Yaskawa INFORM job: A_ROOF_UPPER_0614_2_PAINT_60.JBI

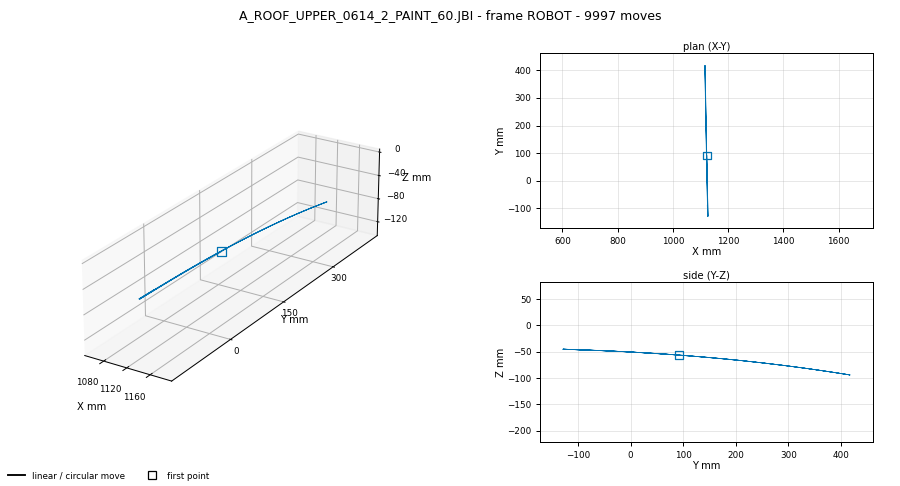
[picture p0: tool path of A_ROOF_UPPER_0614_2_PAINT_60.JBI in frame ROBOT, 9997 of 9997 moves have a stored position in this frame; points joined in program order, loops and branches not executed]
/JOB
//NAME A_ROOF_UPPER_0614_2_PAINT60
//POS
///NPOS 9997,0,0,0,0,0
///TOOL 1
///USER 0
///POSTYPE ROBOT
///RECTAN
///RCONF 1,0,0,0,0,0,0,0,0,0,0,0,0,0,0,0,0,0,0,0,0,0,0,0
C00000=1122.941,91.660,-56.179,-179.955,7.882,149.484
C00001=1122.946,91.411,-56.161,-179.956,7.878,149.483
C00002=1122.951,91.162,-56.142,-179.958,7.874,149.483
C00003=1122.955,90.913,-56.124,-179.959,7.870,149.482
C00004=1122.960,90.663,-56.106,-179.961,7.866,149.482
C00005=1122.965,90.414,-56.088,-179.962,7.862,149.481
C00006=1122.969,90.199,-56.073,-179.963,7.859,149.481
C00007=1122.974,89.984,-56.057,-179.965,7.855,149.480
C00008=1122.978,89.770,-56.041,-179.966,7.852,149.480
C00009=1122.982,89.556,-56.025,-179.967,7.849,149.480
C00010=1122.986,89.341,-56.010,-179.969,7.845,149.479
C00011=1122.990,89.126,-55.995,-179.970,7.842,149.479
C00012=1122.994,88.912,-55.978,-179.971,7.839,149.478
C00013=1122.998,88.697,-55.963,-179.972,7.835,149.478
C00014=1123.004,88.448,-55.944,-179.974,7.831,149.478
C00015=1123.009,88.199,-55.926,-179.975,7.828,149.477
C00016=1123.013,87.950,-55.908,-179.976,7.824,149.477
C00017=1123.018,87.700,-55.891,-179.978,7.820,149.476
C00018=1123.023,87.450,-55.872,-179.979,7.816,149.476
C00019=1123.028,87.201,-55.854,-179.980,7.812,149.475
C00020=1123.033,86.952,-55.836,-179.981,7.809,149.475
C00021=1123.037,86.703,-55.818,-179.983,7.805,149.474
C00022=1123.042,86.454,-55.800,-179.984,7.800,149.474
C00023=1123.048,86.204,-55.783,-179.986,7.797,149.473
C00024=1123.052,85.955,-55.765,-179.987,7.793,149.473
C00025=1123.057,85.706,-55.747,-179.988,7.789,149.472
C00026=1123.062,85.456,-55.729,-179.989,7.785,149.472
C00027=1123.067,85.207,-55.711,-179.991,7.781,149.471
C00028=1123.072,84.957,-55.693,-179.992,7.778,149.471
C00029=1123.076,84.708,-55.675,-179.993,7.774,149.470
C00030=1123.081,84.459,-55.657,-179.995,7.770,149.470
C00031=1123.086,84.210,-55.639,-179.996,7.766,149.469
C00032=1123.091,83.960,-55.622,-179.997,7.763,149.469
C00033=1123.096,83.711,-55.604,-179.998,7.759,149.468
C00034=1123.101,83.462,-55.586,-180.000,7.755,149.468
C00035=1123.105,83.213,-55.568,180.000,7.751,149.467
C00036=1123.110,82.964,-55.550,179.998,7.747,149.466
C00037=1123.116,82.714,-55.533,179.997,7.743,149.466
C00038=1123.120,82.465,-55.515,179.996,7.740,149.465
C00039=1123.125,82.216,-55.497,179.995,7.736,149.465
C00040=1123.130,81.966,-55.479,179.994,7.732,149.464
C00041=1123.136,81.717,-55.462,179.993,7.728,149.464
C00042=1123.140,81.467,-55.443,179.991,7.725,149.463
C00043=1123.145,81.217,-55.425,179.991,7.721,149.463
C00044=1123.150,80.968,-55.407,179.989,7.717,149.462
C00045=1123.154,80.719,-55.391,179.988,7.714,149.462
C00046=1123.159,80.470,-55.373,179.987,7.710,149.461
C00047=1123.164,80.220,-55.355,179.986,7.705,149.461
C00048=1123.169,79.971,-55.338,179.985,7.702,149.460
C00049=1123.174,79.722,-55.320,179.984,7.698,149.460
C00050=1123.179,79.472,-55.302,179.983,7.695,149.459
C00051=1123.183,79.223,-55.285,179.982,7.691,149.459
C00052=1123.188,78.974,-55.267,179.981,7.687,149.458
C00053=1123.193,78.724,-55.249,179.979,7.683,149.457
C00054=1123.199,78.475,-55.232,179.979,7.680,149.457
C00055=1123.204,78.226,-55.214,179.977,7.676,149.456
C00056=1123.209,77.977,-55.197,179.977,7.672,149.456
C00057=1123.213,77.728,-55.179,179.975,7.668,149.455
C00058=1123.218,77.478,-55.161,179.975,7.665,149.455
C00059=1123.224,77.229,-55.144,179.974,7.661,149.454
C00060=1123.228,76.979,-55.126,179.973,7.658,149.454
C00061=1123.233,76.730,-55.110,179.972,7.654,149.453
C00062=1123.237,76.515,-55.094,179.971,7.650,149.453
C00063=1123.241,76.300,-55.079,179.970,7.647,149.452
C00064=1123.245,76.086,-55.063,179.968,7.643,149.452
C00065=1123.250,75.871,-55.049,179.967,7.640,149.451
C00066=1123.255,75.656,-55.034,179.966,7.637,149.451
C00067=1123.258,75.442,-55.019,179.964,7.633,149.451
C00068=1123.262,75.227,-55.004,179.963,7.630,149.450
C00069=1123.266,75.012,-54.989,179.962,7.626,149.450
C00070=1123.272,74.763,-54.971,179.960,7.622,149.449
C00071=1123.276,74.514,-54.955,179.959,7.618,149.449
C00072=1123.282,74.264,-54.937,179.958,7.615,149.448
C00073=1123.287,74.015,-54.919,179.956,7.611,149.448
C00074=1123.291,73.765,-54.903,179.955,7.607,149.447
C00075=1123.296,73.516,-54.885,179.954,7.603,149.447
C00076=1123.301,73.267,-54.867,179.952,7.599,149.446
C00077=1123.305,73.018,-54.850,179.950,7.595,149.446
C00078=1123.311,72.768,-54.833,179.949,7.591,149.445
C00079=1123.316,72.519,-54.816,179.948,7.587,149.445
C00080=1123.321,72.270,-54.798,179.946,7.583,149.444
C00081=1123.326,72.020,-54.781,179.945,7.579,149.444
C00082=1123.330,71.771,-54.765,179.944,7.575,149.443
C00083=1123.335,71.521,-54.747,179.942,7.571,149.443
C00084=1123.340,71.272,-54.729,179.940,7.567,149.442
C00085=1123.345,71.022,-54.713,179.939,7.563,149.442
C00086=1123.350,70.774,-54.695,179.938,7.559,149.441
C00087=1123.355,70.524,-54.678,179.936,7.555,149.441
C00088=1123.360,70.274,-54.661,179.935,7.551,149.441
C00089=1123.365,70.025,-54.644,179.933,7.547,149.440
C00090=1123.369,69.776,-54.626,179.932,7.543,149.439
C00091=1123.375,69.527,-54.610,179.930,7.539,149.439
C00092=1123.380,69.277,-54.593,179.929,7.535,149.439
C00093=1123.385,69.027,-54.576,179.928,7.532,149.438
C00094=1123.389,68.779,-54.558,179.927,7.528,149.438
C00095=1123.394,68.529,-54.541,179.925,7.524,149.437
C00096=1123.399,68.280,-54.525,179.924,7.519,149.436
C00097=1123.405,68.030,-54.507,179.922,7.516,149.436
C00098=1123.409,67.781,-54.491,179.921,7.512,149.436
C00099=1123.414,67.531,-54.473,179.919,7.508,149.435
C00100=1123.419,67.283,-54.456,179.918,7.503,149.435
C00101=1123.424,67.033,-54.439,179.917,7.500,149.434
C00102=1123.429,66.783,-54.422,179.915,7.496,149.434
C00103=1123.433,66.534,-54.406,179.914,7.491,149.433
C00104=1123.439,66.285,-54.389,179.912,7.487,149.433
C00105=1123.444,66.035,-54.372,179.911,7.484,149.432
C00106=1123.449,65.786,-54.355,179.910,7.479,149.432
C00107=1123.453,65.536,-54.338,179.908,7.475,149.431
C00108=1123.459,65.287,-54.321,179.907,7.471,149.431
C00109=1123.464,65.038,-54.305,179.905,7.467,149.430
C00110=1123.468,64.788,-54.288,179.904,7.463,149.430
C00111=1123.473,64.538,-54.271,179.903,7.460,149.429
C00112=1123.478,64.289,-54.255,179.902,7.456,149.429
C00113=1123.483,64.040,-54.238,179.900,7.452,149.428
C00114=1123.488,63.790,-54.221,179.899,7.448,149.428
C00115=1123.493,63.541,-54.204,179.898,7.444,149.427
C00116=1123.498,63.292,-54.188,179.896,7.440,149.427
C00117=1123.503,63.042,-54.170,179.894,7.436,149.426
C00118=1123.507,62.828,-54.156,179.893,7.432,149.426
C00119=1123.511,62.613,-54.141,179.892,7.429,149.425
C00120=1123.515,62.398,-54.127,179.891,7.425,149.425
C00121=1123.520,62.183,-54.113,179.890,7.421,149.424
C00122=1123.524,61.968,-54.099,179.889,7.418,149.424
C00123=1123.529,61.754,-54.084,179.888,7.415,149.423
C00124=1123.532,61.539,-54.070,179.886,7.411,149.423
C00125=1123.537,61.325,-54.055,179.885,7.408,149.422
C00126=1123.542,61.075,-54.039,179.884,7.404,149.422
C00127=1123.546,60.826,-54.022,179.883,7.400,149.421
C00128=1123.552,60.576,-54.006,179.881,7.396,149.421
C00129=1123.557,60.326,-53.989,179.880,7.392,149.421
C00130=1123.561,60.077,-53.973,179.879,7.388,149.420
C00131=1123.566,59.828,-53.956,179.877,7.384,149.419
C00132=1123.572,59.578,-53.939,179.875,7.380,149.419
C00133=1123.577,59.329,-53.923,179.874,7.376,149.418
C00134=1123.581,59.080,-53.907,179.873,7.372,149.418
C00135=1123.586,58.830,-53.890,179.872,7.368,149.417
C00136=1123.592,58.581,-53.873,179.870,7.364,149.417
C00137=1123.596,58.331,-53.856,179.869,7.359,149.416
C00138=1123.602,58.082,-53.841,179.868,7.356,149.416
C00139=1123.606,57.833,-53.824,179.867,7.352,149.415
C00140=1123.611,57.584,-53.808,179.865,7.348,149.415
C00141=1123.617,57.333,-53.791,179.864,7.344,149.414
C00142=1123.621,57.084,-53.775,179.863,7.340,149.414
C00143=1123.626,56.835,-53.758,179.861,7.336,149.413
C00144=1123.631,56.585,-53.742,179.860,7.332,149.413
C00145=1123.636,56.336,-53.726,179.859,7.328,149.412
C00146=1123.641,56.087,-53.709,179.857,7.324,149.412
C00147=1123.646,55.837,-53.694,179.856,7.320,149.411
C00148=1123.651,55.588,-53.677,179.854,7.316,149.411
C00149=1123.656,55.339,-53.660,179.853,7.311,149.410
C00150=1123.661,55.089,-53.644,179.852,7.307,149.410
C00151=1123.666,54.840,-53.628,179.851,7.303,149.409
C00152=1123.671,54.590,-53.611,179.849,7.299,149.409
C00153=1123.676,54.341,-53.596,179.848,7.295,149.408
C00154=1123.680,54.091,-53.579,179.846,7.291,149.407
C00155=1123.686,53.842,-53.564,179.846,7.287,149.407
C00156=1123.690,53.593,-53.547,179.844,7.284,149.406
C00157=1123.696,53.343,-53.531,179.843,7.279,149.406
C00158=1123.700,53.094,-53.515,179.842,7.275,149.405
C00159=1123.706,52.844,-53.499,179.841,7.271,149.405
C00160=1123.711,52.595,-53.482,179.839,7.267,149.404
C00161=1123.716,52.345,-53.466,179.838,7.263,149.404
C00162=1123.721,52.096,-53.450,179.836,7.259,149.403
C00163=1123.726,51.846,-53.434,179.835,7.255,149.403
C00164=1123.731,51.597,-53.417,179.834,7.251,149.402
C00165=1123.736,51.347,-53.402,179.833,7.246,149.401
C00166=1123.741,51.099,-53.385,179.831,7.242,149.401
C00167=1123.746,50.848,-53.369,179.830,7.238,149.400
C00168=1123.751,50.599,-53.354,179.828,7.234,149.400
C00169=1123.756,50.350,-53.337,179.827,7.230,149.399
C00170=1123.760,50.100,-53.322,179.826,7.226,149.399
C00171=1123.765,49.851,-53.305,179.825,7.222,149.398
C00172=1123.770,49.602,-53.290,179.824,7.217,149.398
C00173=1123.776,49.352,-53.274,179.823,7.214,149.397
C00174=1123.779,49.137,-53.260,179.821,7.210,149.397
C00175=1123.784,48.923,-53.246,179.821,7.207,149.396
C00176=1123.788,48.707,-53.233,179.819,7.203,149.396
C00177=1123.793,48.493,-53.219,179.818,7.200,149.395
C00178=1123.797,48.278,-53.205,179.817,7.197,149.395
C00179=1123.801,48.063,-53.192,179.816,7.192,149.394
C00180=1123.805,47.848,-53.178,179.815,7.189,149.394
C00181=1123.810,47.633,-53.163,179.814,7.185,149.393
C00182=1123.814,47.384,-53.148,179.813,7.181,149.393
C00183=1123.820,47.134,-53.133,179.811,7.177,149.392
C00184=1123.824,46.884,-53.117,179.810,7.173,149.392
C00185=1123.830,46.635,-53.101,179.809,7.170,149.391
C00186=1123.835,46.386,-53.085,179.808,7.165,149.390
C00187=1123.840,46.136,-53.069,179.807,7.161,149.390
C00188=1123.845,45.887,-53.053,179.805,7.157,149.389
C00189=1123.849,45.638,-53.038,179.804,7.153,149.389
C00190=1123.854,45.388,-53.022,179.803,7.149,149.388
C00191=1123.860,45.139,-53.006,179.802,7.145,149.388
C00192=1123.865,44.889,-52.991,179.801,7.140,149.387
C00193=1123.870,44.639,-52.975,179.800,7.136,149.386
C00194=1123.874,44.390,-52.960,179.798,7.132,149.386
C00195=1123.880,44.141,-52.943,179.797,7.128,149.385
C00196=1123.884,43.891,-52.927,179.796,7.124,149.385
C00197=1123.890,43.642,-52.912,179.794,7.120,149.384
C00198=1123.895,43.392,-52.896,179.793,7.115,149.384
C00199=1123.900,43.143,-52.881,179.792,7.111,149.383
C00200=1123.904,42.893,-52.865,179.791,7.107,149.383
C00201=1123.910,42.644,-52.850,179.789,7.103,149.382
C00202=1123.915,42.395,-52.835,179.788,7.098,149.381
C00203=1123.919,42.145,-52.819,179.787,7.095,149.381
C00204=1123.925,41.895,-52.803,179.786,7.090,149.380
C00205=1123.930,41.646,-52.788,179.785,7.086,149.380
C00206=1123.935,41.397,-52.773,179.784,7.082,149.379
C00207=1123.939,41.147,-52.756,179.782,7.078,149.378
C00208=1123.945,40.898,-52.740,179.781,7.073,149.378
C00209=1123.949,40.649,-52.725,179.780,7.069,149.377
C00210=1123.955,40.399,-52.710,179.778,7.065,149.377
C00211=1123.960,40.149,-52.695,179.777,7.061,149.376
C00212=1123.964,39.899,-52.680,179.777,7.057,149.375
C00213=1123.970,39.650,-52.664,179.776,7.053,149.375
C00214=1123.975,39.401,-52.648,179.775,7.049,149.374
C00215=1123.980,39.152,-52.633,179.773,7.045,149.374
C00216=1123.985,38.901,-52.617,179.772,7.040,149.373
C00217=1123.990,38.652,-52.602,179.771,7.036,149.372
C00218=1123.995,38.403,-52.587,179.770,7.032,149.372
C00219=1124.000,38.154,-52.571,179.768,7.028,149.371
C00220=1124.005,37.904,-52.556,179.767,7.024,149.371
C00221=1124.010,37.655,-52.541,179.766,7.019,149.370
C00222=1124.015,37.404,-52.525,179.765,7.015,149.369
C00223=1124.020,37.155,-52.510,179.764,7.011,149.369
C00224=1124.025,36.906,-52.495,179.763,7.006,149.368
C00225=1124.030,36.657,-52.480,179.762,7.002,149.368
C00226=1124.035,36.407,-52.464,179.760,6.998,149.367
C00227=1124.041,36.158,-52.449,179.759,6.994,149.366
C00228=1124.046,35.908,-52.434,179.758,6.990,149.366
C00229=1124.050,35.658,-52.418,179.757,6.985,149.365
C00230=1124.054,35.443,-52.406,179.756,6.981,149.365
C00231=1124.059,35.229,-52.393,179.755,6.978,149.364
C00232=1124.063,35.014,-52.379,179.754,6.975,149.364
C00233=1124.068,34.799,-52.366,179.753,6.970,149.363
C00234=1124.072,34.584,-52.353,179.752,6.967,149.362
C00235=1124.076,34.369,-52.340,179.751,6.963,149.362
C00236=1124.081,34.154,-52.327,179.750,6.960,149.361
C00237=1124.085,33.939,-52.315,179.749,6.955,149.361
C00238=1124.090,33.690,-52.299,179.748,6.952,149.360
C00239=1124.095,33.440,-52.285,179.747,6.947,149.360
C00240=1124.101,33.191,-52.269,179.746,6.943,149.359
C00241=1124.105,32.941,-52.254,179.745,6.939,149.358
C00242=1124.110,32.691,-52.239,179.744,6.934,149.358
C00243=1124.115,32.442,-52.224,179.743,6.930,149.357
C00244=1124.120,32.192,-52.208,179.741,6.926,149.356
C00245=1124.125,31.942,-52.194,179.740,6.921,149.356
C00246=1124.130,31.693,-52.179,179.739,6.917,149.355
C00247=1124.135,31.444,-52.163,179.738,6.913,149.354
C00248=1124.140,31.194,-52.149,179.737,6.908,149.354
C00249=1124.146,30.945,-52.134,179.736,6.904,149.353
C00250=1124.151,30.695,-52.119,179.735,6.900,149.353
C00251=1124.155,30.446,-52.104,179.734,6.895,149.352
C00252=1124.161,30.197,-52.089,179.733,6.891,149.351
C00253=1124.166,29.947,-52.074,179.732,6.887,149.351
C00254=1124.171,29.698,-52.059,179.731,6.883,149.350
C00255=1124.176,29.448,-52.045,179.730,6.878,149.349
C00256=1124.181,29.199,-52.030,179.729,6.874,149.349
C00257=1124.186,28.949,-52.015,179.728,6.870,149.348
C00258=1124.191,28.700,-52.000,179.727,6.865,149.347
C00259=1124.196,28.450,-51.985,179.726,6.861,149.347
C00260=1124.201,28.201,-51.970,179.725,6.857,149.346
C00261=1124.206,27.951,-51.956,179.723,6.852,149.345
C00262=1124.211,27.701,-51.941,179.722,6.848,149.345
C00263=1124.216,27.452,-51.926,179.721,6.844,149.344
C00264=1124.221,27.202,-51.911,179.720,6.839,149.343
C00265=1124.226,26.953,-51.896,179.719,6.835,149.343
C00266=1124.231,26.703,-51.882,179.718,6.831,149.342
C00267=1124.236,26.454,-51.867,179.718,6.826,149.341
C00268=1124.241,26.204,-51.852,179.717,6.822,149.341
C00269=1124.246,25.954,-51.838,179.716,6.817,149.340
C00270=1124.251,25.705,-51.823,179.714,6.813,149.339
C00271=1124.257,25.455,-51.808,179.713,6.809,149.339
C00272=1124.262,25.206,-51.794,179.712,6.804,149.338
C00273=1124.266,24.956,-51.779,179.711,6.800,149.337
C00274=1124.271,24.707,-51.765,179.710,6.796,149.337
C00275=1124.277,24.458,-51.751,179.710,6.791,149.336
C00276=1124.282,24.208,-51.735,179.709,6.787,149.335
C00277=1124.287,23.959,-51.721,179.707,6.782,149.335
C00278=1124.292,23.709,-51.707,179.706,6.777,149.334
C00279=1124.297,23.460,-51.692,179.705,6.773,149.333
C00280=1124.302,23.210,-51.677,179.704,6.768,149.332
C00281=1124.307,22.960,-51.662,179.703,6.764,149.332
C00282=1124.312,22.710,-51.648,179.702,6.760,149.331
C00283=1124.317,22.461,-51.633,179.701,6.755,149.330
C00284=1124.322,22.212,-51.619,179.700,6.751,149.330
C00285=1124.328,21.963,-51.605,179.700,6.746,149.329
C00286=1124.332,21.748,-51.592,179.699,6.743,149.328
C00287=1124.336,21.532,-51.580,179.698,6.739,149.328
C00288=1124.341,21.317,-51.567,179.697,6.735,149.327
C00289=1124.345,21.102,-51.556,179.696,6.731,149.327
C00290=1124.349,20.886,-51.542,179.696,6.728,149.326
C00291=1124.353,20.672,-51.530,179.694,6.724,149.325
C00292=1124.358,20.456,-51.518,179.693,6.719,149.325
C00293=1124.362,20.242,-51.505,179.693,6.716,149.324
C00294=1124.367,19.993,-51.491,179.692,6.711,149.323
C00295=1124.372,19.743,-51.477,179.691,6.707,149.323
C00296=1124.378,19.493,-51.462,179.690,6.702,149.322
C00297=1124.383,19.243,-51.448,179.689,6.698,149.321
C00298=1124.388,18.993,-51.434,179.688,6.693,149.320
C00299=1124.393,18.744,-51.420,179.687,6.689,149.320
C00300=1124.398,18.495,-51.405,179.686,6.684,149.319
C00301=1124.403,18.245,-51.391,179.685,6.679,149.318
C00302=1124.408,17.995,-51.377,179.684,6.675,149.318
C00303=1124.413,17.746,-51.363,179.683,6.671,149.317
C00304=1124.419,17.497,-51.349,179.683,6.666,149.316
C00305=1124.424,17.247,-51.334,179.682,6.662,149.315
C00306=1124.429,16.997,-51.320,179.681,6.657,149.315
C00307=1124.434,16.747,-51.306,179.680,6.652,149.314
C00308=1124.439,16.498,-51.292,179.679,6.648,149.313
C00309=1124.444,16.249,-51.278,179.678,6.643,149.312
C00310=1124.449,15.999,-51.263,179.677,6.638,149.312
C00311=1124.454,15.749,-51.249,179.676,6.634,149.311
C00312=1124.460,15.500,-51.235,179.675,6.629,149.310
C00313=1124.465,15.251,-51.221,179.674,6.625,149.310
C00314=1124.469,15.001,-51.207,179.673,6.620,149.309
C00315=1124.474,14.751,-51.193,179.672,6.616,149.308
C00316=1124.479,14.502,-51.179,179.672,6.611,149.307
C00317=1124.484,14.253,-51.165,179.671,6.607,149.306
C00318=1124.489,14.003,-51.150,179.670,6.602,149.306
C00319=1124.494,13.753,-51.136,179.669,6.597,149.305
C00320=1124.500,13.504,-51.123,179.668,6.592,149.304
C00321=1124.505,13.254,-51.109,179.667,6.588,149.303
C00322=1124.510,13.004,-51.094,179.667,6.583,149.303
C00323=1124.515,12.755,-51.081,179.665,6.579,149.302
C00324=1124.520,12.506,-51.067,179.665,6.574,149.301
C00325=1124.525,12.256,-51.053,179.664,6.570,149.300
C00326=1124.531,12.007,-51.039,179.663,6.565,149.299
C00327=1124.535,11.757,-51.025,179.662,6.560,149.299
C00328=1124.540,11.507,-51.011,179.661,6.555,149.298
C00329=1124.546,11.258,-50.997,179.661,6.551,149.297
C00330=1124.551,11.008,-50.984,179.660,6.546,149.296
C00331=1124.555,10.758,-50.970,179.659,6.542,149.296
C00332=1124.561,10.509,-50.956,179.658,6.537,149.295
C00333=1124.566,10.260,-50.941,179.657,6.533,149.294
C00334=1124.571,10.009,-50.928,179.656,6.527,149.293
C00335=1124.576,9.761,-50.915,179.655,6.523,149.292
C00336=1124.581,9.511,-50.900,179.655,6.518,149.292
C00337=1124.587,9.261,-50.887,179.654,6.513,149.291
C00338=1124.592,9.012,-50.873,179.653,6.509,149.290
C00339=1124.596,8.762,-50.859,179.653,6.504,149.289
C00340=1124.602,8.513,-50.846,179.651,6.499,149.288
C00341=1124.607,8.263,-50.832,179.650,6.494,149.288
C00342=1124.611,8.048,-50.820,179.650,6.491,149.287
C00343=1124.616,7.833,-50.809,179.650,6.487,149.286
C00344=1124.621,7.617,-50.796,179.650,6.482,149.285
C00345=1124.625,7.402,-50.785,179.649,6.479,149.285
C00346=1124.629,7.187,-50.773,179.649,6.475,149.284
C00347=1124.633,6.972,-50.761,179.649,6.471,149.283
C00348=1124.637,6.757,-50.749,179.648,6.467,149.282
C00349=1124.643,6.542,-50.737,179.647,6.463,149.282
C00350=1124.647,6.292,-50.724,179.647,6.459,149.281
C00351=1124.652,6.042,-50.710,179.647,6.455,149.280
C00352=1124.658,5.793,-50.697,179.646,6.450,149.279
C00353=1124.662,5.543,-50.683,179.646,6.445,149.278
C00354=1124.668,5.294,-50.670,179.645,6.441,149.277
C00355=1124.673,5.044,-50.655,179.645,6.436,149.276
C00356=1124.678,4.795,-50.643,179.645,6.432,149.276
C00357=1124.683,4.545,-50.629,179.644,6.428,149.275
C00358=1124.689,4.295,-50.615,179.643,6.423,149.274
C00359=1124.693,4.046,-50.602,179.643,6.418,149.273
C00360=1124.699,3.796,-50.589,179.642,6.413,149.272
C00361=1124.703,3.547,-50.575,179.642,6.410,149.271
C00362=1124.709,3.297,-50.562,179.642,6.405,149.270
C00363=1124.714,3.048,-50.547,179.641,6.400,149.270
C00364=1124.719,2.798,-50.535,179.640,6.396,149.269
C00365=1124.724,2.549,-50.520,179.640,6.391,149.268
C00366=1124.729,2.299,-50.508,179.640,6.387,149.267
C00367=1124.734,2.049,-50.494,179.639,6.382,149.266
C00368=1124.740,1.800,-50.480,179.638,6.378,149.266
C00369=1124.745,1.550,-50.467,179.638,6.373,149.265
C00370=1124.750,1.301,-50.454,179.637,6.369,149.264
C00371=1124.755,1.051,-50.441,179.637,6.364,149.263
C00372=1124.761,0.801,-50.427,179.637,6.360,149.262
C00373=1124.765,0.552,-50.414,179.636,6.356,149.261
C00374=1124.771,0.302,-50.401,179.635,6.351,149.261
C00375=1124.775,0.052,-50.388,179.635,6.346,149.260
C00376=1124.781,-0.197,-50.374,179.634,6.341,149.259
C00377=1124.785,-0.447,-50.361,179.633,6.337,149.258
C00378=1124.791,-0.696,-50.347,179.633,6.333,149.257
C00379=1124.795,-0.946,-50.334,179.633,6.328,149.256
C00380=1124.801,-1.195,-50.321,179.632,6.324,149.256
C00381=1124.806,-1.445,-50.308,179.631,6.319,149.255
C00382=1124.811,-1.694,-50.294,179.631,6.315,149.254
C00383=1124.816,-1.944,-50.281,179.630,6.310,149.253
C00384=1124.822,-2.194,-50.268,179.629,6.306,149.252
C00385=1124.827,-2.443,-50.255,179.629,6.302,149.252
C00386=1124.832,-2.692,-50.241,179.629,6.297,149.251
C00387=1124.837,-2.942,-50.228,179.628,6.292,149.250
C00388=1124.843,-3.192,-50.215,179.627,6.288,149.249
C00389=1124.847,-3.442,-50.202,179.627,6.283,149.248
C00390=1124.853,-3.692,-50.189,179.626,6.278,149.247
C00391=1124.858,-3.940,-50.175,179.625,6.274,149.247
C00392=1124.862,-4.190,-50.162,179.624,6.269,149.246
C00393=1124.868,-4.440,-50.149,179.624,6.265,149.245
C00394=1124.873,-4.690,-50.136,179.624,6.261,149.244
C00395=1124.879,-4.940,-50.123,179.623,6.256,149.243
C00396=1124.884,-5.189,-50.110,179.623,6.252,149.242
C00397=1124.888,-5.438,-50.097,179.622,6.247,149.242
C00398=1124.893,-5.654,-50.086,179.621,6.243,149.241
C00399=1124.897,-5.869,-50.075,179.621,6.239,149.240
C00400=1124.902,-6.085,-50.064,179.620,6.236,149.240
C00401=1124.906,-6.299,-50.052,179.619,6.231,149.239
C00402=1124.911,-6.515,-50.041,179.619,6.228,149.238
C00403=1124.915,-6.731,-50.030,179.618,6.223,149.238
C00404=1124.920,-6.945,-50.018,179.618,6.219,149.237
C00405=1124.924,-7.161,-50.007,179.618,6.216,149.236
C00406=1124.929,-7.410,-49.995,179.617,6.211,149.235
C00407=1124.934,-7.660,-49.982,179.616,6.207,149.235
C00408=1124.940,-7.910,-49.969,179.616,6.202,149.234
C00409=1124.945,-8.159,-49.956,179.615,6.198,149.233
C00410=1124.950,-8.409,-49.943,179.614,6.193,149.232
C00411=1124.955,-8.659,-49.930,179.614,6.188,149.231
C00412=1124.961,-8.908,-49.917,179.613,6.184,149.231
C00413=1124.966,-9.158,-49.905,179.612,6.179,149.230
C00414=1124.970,-9.408,-49.892,179.612,6.174,149.229
C00415=1124.976,-9.657,-49.878,179.611,6.170,149.228
C00416=1124.981,-9.906,-49.866,179.610,6.165,149.227
C00417=1124.986,-10.157,-49.853,179.610,6.161,149.226
C00418=1124.991,-10.406,-49.840,179.609,6.156,149.226
C00419=1124.997,-10.655,-49.827,179.608,6.152,149.225
C00420=1125.002,-10.905,-49.814,179.608,6.147,149.224
C00421=1125.006,-11.155,-49.801,179.607,6.142,149.223
C00422=1125.011,-11.404,-49.789,179.606,6.138,149.222
C00423=1125.017,-11.654,-49.776,179.606,6.133,149.221
C00424=1125.022,-11.903,-49.763,179.605,6.129,149.221
C00425=1125.027,-12.153,-49.750,179.604,6.124,149.220
C00426=1125.032,-12.403,-49.738,179.604,6.119,149.219
C00427=1125.037,-12.652,-49.726,179.603,6.115,149.218
C00428=1125.043,-12.902,-49.713,179.602,6.110,149.217
C00429=1125.048,-13.152,-49.699,179.602,6.105,149.217
C00430=1125.053,-13.401,-49.687,179.601,6.101,149.216
C00431=1125.058,-13.651,-49.674,179.600,6.096,149.215
C00432=1125.064,-13.901,-49.662,179.600,6.092,149.214
C00433=1125.069,-14.150,-49.650,179.599,6.087,149.213
C00434=1125.073,-14.400,-49.637,179.598,6.082,149.213
C00435=1125.078,-14.649,-49.624,179.597,6.077,149.212
C00436=1125.084,-14.899,-49.611,179.596,6.073,149.211
C00437=1125.090,-15.149,-49.599,179.596,6.068,149.210
C00438=1125.095,-15.398,-49.587,179.595,6.063,149.209
C00439=1125.100,-15.647,-49.574,179.595,6.058,149.208
C00440=1125.104,-15.897,-49.561,179.594,6.054,149.208
C00441=1125.110,-16.147,-49.549,179.593,6.049,149.207
C00442=1125.115,-16.397,-49.536,179.593,6.045,149.206
C00443=1125.120,-16.646,-49.524,179.592,6.040,149.205
C00444=1125.125,-16.896,-49.512,179.591,6.035,149.204
C00445=1125.131,-17.145,-49.499,179.590,6.030,149.203
C00446=1125.135,-17.395,-49.486,179.589,6.026,149.203
C00447=1125.141,-17.645,-49.475,179.589,6.021,149.202
C00448=1125.146,-17.895,-49.461,179.588,6.016,149.201
C00449=1125.152,-18.144,-49.449,179.588,6.011,149.200
C00450=1125.157,-18.394,-49.437,179.586,6.006,149.200
C00451=1125.162,-18.643,-49.424,179.586,6.002,149.199
C00452=1125.168,-18.893,-49.412,179.585,5.997,149.198
C00453=1125.173,-19.143,-49.400,179.584,5.993,149.197
C00454=1125.176,-19.358,-49.389,179.584,5.988,149.196
C00455=1125.181,-19.573,-49.379,179.583,5.984,149.195
C00456=1125.186,-19.789,-49.368,179.582,5.980,149.195
C00457=1125.190,-20.004,-49.358,179.581,5.976,149.194
C00458=1125.194,-20.219,-49.346,179.581,5.972,149.193
C00459=1125.199,-20.434,-49.336,179.580,5.967,149.193
C00460=1125.203,-20.650,-49.325,179.580,5.964,149.192
C00461=1125.208,-20.865,-49.315,179.579,5.959,149.191
C00462=1125.214,-21.115,-49.303,179.579,5.955,149.190
C00463=1125.218,-21.364,-49.291,179.578,5.949,149.189
C00464=1125.224,-21.614,-49.279,179.577,5.944,149.189
C00465=1125.229,-21.864,-49.266,179.576,5.940,149.188
C00466=1125.234,-22.114,-49.254,179.576,5.935,149.187
C00467=1125.239,-22.363,-49.242,179.575,5.930,149.186
C00468=1125.245,-22.613,-49.230,179.574,5.925,149.185
C00469=1125.250,-22.862,-49.217,179.574,5.920,149.184
C00470=1125.255,-23.112,-49.205,179.573,5.916,149.184
C00471=1125.261,-23.362,-49.193,179.572,5.910,149.183
C00472=1125.266,-23.611,-49.181,179.571,5.906,149.182
C00473=1125.271,-23.861,-49.169,179.571,5.901,149.181
C00474=1125.276,-24.110,-49.157,179.569,5.895,149.180
C00475=1125.281,-24.360,-49.145,179.569,5.891,149.179
C00476=1125.286,-24.610,-49.133,179.568,5.886,149.179
C00477=1125.292,-24.859,-49.121,179.567,5.881,149.178
C00478=1125.297,-25.109,-49.109,179.566,5.876,149.177
C00479=1125.302,-25.359,-49.097,179.566,5.871,149.176
C00480=1125.307,-25.608,-49.085,179.565,5.866,149.175
C00481=1125.312,-25.858,-49.073,179.564,5.861,149.174
C00482=1125.318,-26.108,-49.061,179.565,5.857,149.173
C00483=1125.323,-26.357,-49.048,179.565,5.853,149.172
C00484=1125.328,-26.607,-49.037,179.566,5.849,149.171
C00485=1125.333,-26.857,-49.025,179.567,5.845,149.170
C00486=1125.338,-27.107,-49.013,179.568,5.841,149.169
C00487=1125.344,-27.356,-49.001,179.569,5.837,149.168
C00488=1125.349,-27.606,-48.989,179.570,5.833,149.166
C00489=1125.354,-27.856,-48.978,179.571,5.829,149.165
C00490=1125.359,-28.105,-48.965,179.571,5.825,149.164
C00491=1125.364,-28.355,-48.953,179.571,5.821,149.163
C00492=1125.370,-28.605,-48.941,179.572,5.816,149.162
C00493=1125.374,-28.855,-48.930,179.573,5.813,149.161
C00494=1125.379,-29.104,-48.917,179.573,5.809,149.160
C00495=1125.385,-29.354,-48.905,179.574,5.805,149.159
C00496=1125.390,-29.604,-48.894,179.574,5.801,149.158
C00497=1125.395,-29.854,-48.882,179.575,5.796,149.157
C00498=1125.401,-30.102,-48.870,179.575,5.792,149.156
C00499=1125.406,-30.352,-48.858,179.575,5.789,149.155
C00500=1125.412,-30.602,-48.846,179.576,5.784,149.154
C00501=1125.416,-30.852,-48.835,179.575,5.779,149.153
C00502=1125.422,-31.102,-48.823,179.575,5.775,149.152
C00503=1125.427,-31.351,-48.810,179.576,5.772,149.151
C00504=1125.432,-31.601,-48.799,179.576,5.768,149.150
C00505=1125.437,-31.850,-48.787,179.576,5.762,149.149
C00506=1125.442,-32.100,-48.775,179.576,5.759,149.148
C00507=1125.448,-32.350,-48.764,179.575,5.754,149.147
C00508=1125.452,-32.600,-48.752,179.576,5.750,149.147
C00509=1125.458,-32.849,-48.740,179.575,5.745,149.146
C00510=1125.462,-33.065,-48.730,179.575,5.742,149.145
C00511=1125.467,-33.280,-48.720,179.574,5.738,149.144
C00512=1125.472,-33.495,-48.710,179.575,5.734,149.143
C00513=1125.476,-33.711,-48.700,179.574,5.730,149.143
C00514=1125.481,-33.926,-48.690,179.573,5.726,149.142
C00515=1125.485,-34.141,-48.680,179.573,5.722,149.141
C00516=1125.490,-34.358,-48.669,179.573,5.719,149.140
C00517=1125.494,-34.572,-48.659,179.572,5.714,149.140
C00518=1125.500,-34.822,-48.647,179.572,5.709,149.139
C00519=1125.504,-35.072,-48.636,179.571,5.705,149.138
C00520=1125.510,-35.322,-48.624,179.570,5.700,149.137
C00521=1125.515,-35.571,-48.613,179.570,5.696,149.136
C00522=1125.521,-35.821,-48.601,179.569,5.691,149.136
C00523=1125.526,-36.071,-48.589,179.569,5.687,149.135
C00524=1125.531,-36.320,-48.578,179.567,5.681,149.134
C00525=1125.536,-36.570,-48.566,179.567,5.677,149.133
C00526=1125.541,-36.820,-48.555,179.566,5.672,149.133
C00527=1125.547,-37.069,-48.544,179.565,5.667,149.132
C00528=1125.552,-37.319,-48.532,179.564,5.662,149.131
C00529=1125.557,-37.569,-48.520,179.563,5.657,149.130
C00530=1125.562,-37.819,-48.508,179.562,5.652,149.129
C00531=1125.567,-38.068,-48.497,179.561,5.647,149.129
C00532=1125.573,-38.317,-48.486,179.559,5.642,149.128
C00533=1125.578,-38.567,-48.474,179.557,5.637,149.127
C00534=1125.583,-38.817,-48.462,179.557,5.632,149.126
C00535=1125.588,-39.067,-48.451,179.556,5.627,149.126
C00536=1125.594,-39.316,-48.440,179.554,5.622,149.125
C00537=1125.599,-39.566,-48.429,179.553,5.616,149.124
C00538=1125.604,-39.816,-48.417,179.551,5.611,149.123
C00539=1125.609,-40.066,-48.406,179.550,5.606,149.123
C00540=1125.615,-40.315,-48.394,179.548,5.601,149.122
C00541=1125.620,-40.565,-48.383,179.547,5.594,149.121
C00542=1125.625,-40.815,-48.371,179.545,5.589,149.121
C00543=1125.631,-41.064,-48.361,179.544,5.584,149.120
C00544=1125.636,-41.314,-48.349,179.541,5.578,149.119
C00545=1125.641,-41.564,-48.338,179.540,5.572,149.118
C00546=1125.646,-41.813,-48.327,179.538,5.566,149.118
C00547=1125.652,-42.063,-48.316,179.537,5.561,149.117
C00548=1125.657,-42.313,-48.304,179.535,5.555,149.116
C00549=1125.661,-42.562,-48.293,179.533,5.549,149.115
C00550=1125.668,-42.812,-48.282,179.532,5.544,149.115
C00551=1125.672,-43.062,-48.271,179.529,5.538,149.114
C00552=1125.678,-43.311,-48.260,179.529,5.533,149.113
C00553=1125.683,-43.561,-48.249,179.529,5.528,149.112
C00554=1125.688,-43.811,-48.238,179.529,5.523,149.111
C00555=1125.694,-44.060,-48.226,179.529,5.519,149.110
C00556=1125.699,-44.310,-48.216,179.529,5.514,149.109
C00557=1125.704,-44.560,-48.204,179.530,5.509,149.108
C00558=1125.709,-44.810,-48.194,179.530,5.504,149.107
C00559=1125.715,-45.060,-48.182,179.530,5.500,149.106
C00560=1125.720,-45.309,-48.171,179.530,5.495,149.105
C00561=1125.725,-45.559,-48.161,179.530,5.490,149.103
C00562=1125.731,-45.809,-48.149,179.531,5.486,149.102
C00563=1125.736,-46.058,-48.139,179.531,5.481,149.101
C00564=1125.741,-46.308,-48.127,179.531,5.477,149.100
C00565=1125.746,-46.558,-48.117,179.531,5.471,149.099
C00566=1125.750,-46.773,-48.107,179.531,5.467,149.098
C00567=1125.756,-46.989,-48.097,179.532,5.463,149.097
C00568=1125.760,-47.204,-48.088,179.532,5.460,149.096
C00569=1125.765,-47.420,-48.078,179.532,5.456,149.095
C00570=1125.769,-47.635,-48.069,179.532,5.452,149.095
C00571=1125.774,-47.851,-48.060,179.532,5.447,149.094
C00572=1125.779,-48.066,-48.050,179.532,5.443,149.093
C00573=1125.783,-48.282,-48.041,179.532,5.439,149.092
C00574=1125.788,-48.531,-48.030,179.533,5.435,149.091
C00575=1125.793,-48.782,-48.019,179.533,5.429,149.090
C00576=1125.798,-49.030,-48.008,179.534,5.425,149.088
C00577=1125.804,-49.281,-47.997,179.533,5.420,149.087
C00578=1125.809,-49.530,-47.986,179.533,5.415,149.086
C00579=1125.814,-49.780,-47.976,179.534,5.411,149.085
C00580=1125.820,-50.029,-47.965,179.533,5.406,149.084
C00581=1125.825,-50.279,-47.954,179.534,5.402,149.083
C00582=1125.830,-50.529,-47.942,179.534,5.397,149.082
C00583=1125.836,-50.779,-47.932,179.534,5.393,149.081
C00584=1125.841,-51.029,-47.921,179.534,5.388,149.080
C00585=1125.846,-51.278,-47.911,179.535,5.382,149.079
C00586=1125.851,-51.528,-47.900,179.535,5.378,149.078
C00587=1125.856,-51.777,-47.889,179.535,5.373,149.077
C00588=1125.862,-52.028,-47.878,179.535,5.369,149.076
C00589=1125.868,-52.277,-47.868,179.536,5.364,149.074
C00590=1125.872,-52.527,-47.856,179.536,5.360,149.074
C00591=1125.878,-52.776,-47.846,179.536,5.355,149.072
C00592=1125.883,-53.026,-47.835,179.536,5.350,149.071
C00593=1125.888,-53.276,-47.825,179.536,5.346,149.070
C00594=1125.893,-53.526,-47.814,179.536,5.340,149.069
C00595=1125.899,-53.775,-47.803,179.537,5.336,149.068
C00596=1125.904,-54.025,-47.792,179.536,5.331,149.067
C00597=1125.910,-54.275,-47.782,179.537,5.327,149.066
C00598=1125.915,-54.525,-47.771,179.537,5.322,149.065
C00599=1125.920,-54.774,-47.760,179.537,5.318,149.064
C00600=1125.925,-55.024,-47.750,179.538,5.313,149.063
C00601=1125.931,-55.274,-47.740,179.538,5.308,149.062
C00602=1125.935,-55.523,-47.728,179.538,5.303,149.060
C00603=1125.941,-55.773,-47.718,179.538,5.298,149.060
C00604=1125.946,-56.023,-47.707,179.539,5.294,149.058
C00605=1125.951,-56.272,-47.697,179.539,5.289,149.057
C00606=1125.957,-56.522,-47.686,179.539,5.285,149.056
C00607=1125.962,-56.772,-47.676,179.539,5.280,149.055
C00608=1125.968,-57.022,-47.666,179.539,5.276,149.054
C00609=1125.972,-57.271,-47.654,179.539,5.271,149.053
C00610=1125.978,-57.521,-47.644,179.539,5.266,149.052
C00611=1125.983,-57.771,-47.633,179.540,5.262,149.051
C00612=1125.988,-58.020,-47.623,179.540,5.257,149.050
C00613=1125.993,-58.271,-47.613,179.540,5.252,149.049
C00614=1125.999,-58.520,-47.602,179.540,5.247,149.048
C00615=1126.004,-58.769,-47.592,179.541,5.243,149.047
C00616=1126.009,-59.019,-47.581,179.541,5.238,149.045
C00617=1126.015,-59.269,-47.571,179.541,5.234,149.045
C00618=1126.020,-59.519,-47.560,179.541,5.229,149.043
C00619=1126.025,-59.768,-47.549,179.542,5.224,149.042
C00620=1126.030,-60.018,-47.539,179.541,5.220,149.041
C00621=1126.036,-60.268,-47.528,179.541,5.215,149.040
C00622=1126.040,-60.483,-47.519,179.541,5.210,149.040
C00623=1126.045,-60.700,-47.511,179.540,5.206,149.039
C00624=1126.050,-60.915,-47.501,179.539,5.201,149.038
C00625=1126.055,-61.131,-47.492,179.538,5.197,149.037
C00626=1126.059,-61.346,-47.483,179.537,5.192,149.037
C00627=1126.064,-61.562,-47.475,179.537,5.188,149.036
C00628=1126.068,-61.777,-47.465,179.536,5.183,149.035
C00629=1126.073,-61.993,-47.456,179.535,5.179,149.034
C00630=1126.078,-62.242,-47.446,179.534,5.173,149.033
C00631=1126.083,-62.492,-47.436,179.533,5.168,149.032
C00632=1126.088,-62.742,-47.426,179.532,5.162,149.032
C00633=1126.094,-62.991,-47.416,179.532,5.157,149.031
C00634=1126.099,-63.242,-47.405,179.531,5.152,149.030
C00635=1126.104,-63.491,-47.395,179.530,5.146,149.029
C00636=1126.110,-63.741,-47.385,179.530,5.141,149.028
C00637=1126.115,-63.991,-47.374,179.529,5.135,149.027
C00638=1126.121,-64.241,-47.364,179.528,5.130,149.026
C00639=1126.126,-64.490,-47.354,179.528,5.125,149.025
C00640=1126.131,-64.740,-47.344,179.527,5.120,149.024
C00641=1126.136,-64.990,-47.333,179.526,5.114,149.023
C00642=1126.142,-65.239,-47.323,179.525,5.109,149.022
C00643=1126.147,-65.490,-47.313,179.524,5.104,149.021
C00644=1126.152,-65.739,-47.304,179.525,5.099,149.020
C00645=1126.157,-65.989,-47.294,179.524,5.093,149.019
C00646=1126.163,-66.238,-47.283,179.523,5.087,149.018
C00647=1126.168,-66.488,-47.273,179.522,5.083,149.017
C00648=1126.174,-66.738,-47.263,179.522,5.077,149.016
C00649=1126.179,-66.987,-47.253,179.521,5.072,149.015
C00650=1126.184,-67.237,-47.243,179.520,5.066,149.014
C00651=1126.189,-67.488,-47.233,179.520,5.062,149.013
C00652=1126.195,-67.737,-47.223,179.520,5.056,149.012
C00653=1126.200,-67.986,-47.213,179.519,5.051,149.011
C00654=1126.206,-68.236,-47.203,179.519,5.045,149.010
C00655=1126.211,-68.486,-47.193,179.518,5.039,149.009
C00656=1126.216,-68.736,-47.183,179.517,5.035,149.008
C00657=1126.221,-68.986,-47.173,179.517,5.029,149.007
C00658=1126.227,-69.235,-47.163,179.517,5.024,149.006
C00659=1126.232,-69.485,-47.153,179.517,5.019,149.005
C00660=1126.238,-69.735,-47.144,179.516,5.013,149.004
C00661=1126.243,-69.985,-47.133,179.516,5.008,149.003
C00662=1126.248,-70.234,-47.123,179.515,5.002,149.002
C00663=1126.253,-70.484,-47.114,179.515,4.997,149.001
C00664=1126.259,-70.734,-47.104,179.514,4.992,149.000
C00665=1126.265,-70.983,-47.094,179.514,4.986,148.999
C00666=1126.269,-71.234,-47.084,179.513,4.981,148.998
C00667=1126.275,-71.483,-47.074,179.513,4.976,148.997
C00668=1126.280,-71.733,-47.064,179.513,4.971,148.996
C00669=1126.286,-71.983,-47.055,179.513,4.965,148.995
C00670=1126.291,-72.232,-47.045,179.513,4.960,148.994
C00671=1126.296,-72.482,-47.035,179.512,4.955,148.993
C00672=1126.302,-72.732,-47.026,179.512,4.949,148.992
C00673=1126.307,-72.981,-47.016,179.512,4.944,148.990
C00674=1126.312,-73.232,-47.006,179.512,4.939,148.990
C00675=1126.318,-73.481,-46.996,179.511,4.933,148.988
C00676=1126.323,-73.731,-46.987,179.511,4.928,148.987
C00677=1126.328,-73.981,-46.977,179.511,4.923,148.986
C00678=1126.333,-74.197,-46.969,179.511,4.919,148.985
C00679=1126.337,-74.412,-46.960,179.511,4.913,148.984
C00680=1126.342,-74.627,-46.952,179.511,4.909,148.983
C00681=1126.347,-74.843,-46.944,179.511,4.905,148.982
C00682=1126.351,-75.059,-46.936,179.510,4.900,148.981
C00683=1126.356,-75.275,-46.927,179.511,4.896,148.980
C00684=1126.361,-75.490,-46.919,179.510,4.891,148.980
C00685=1126.366,-75.706,-46.910,179.510,4.886,148.979
C00686=1126.371,-75.956,-46.901,179.510,4.881,148.977
C00687=1126.376,-76.205,-46.891,179.510,4.876,148.976
C00688=1126.382,-76.455,-46.882,179.510,4.871,148.975
C00689=1126.387,-76.706,-46.872,179.510,4.866,148.974
C00690=1126.392,-76.955,-46.863,179.510,4.860,148.973
C00691=1126.398,-77.205,-46.853,179.510,4.855,148.972
C00692=1126.403,-77.455,-46.844,179.510,4.850,148.971
C00693=1126.408,-77.705,-46.834,179.510,4.845,148.970
C00694=1126.413,-77.954,-46.824,179.510,4.839,148.968
C00695=1126.419,-78.204,-46.815,179.510,4.834,148.967
C00696=1126.424,-78.454,-46.806,179.510,4.829,148.966
C00697=1126.430,-78.703,-46.796,179.511,4.824,148.965
C00698=1126.435,-78.953,-46.787,179.510,4.818,148.964
C00699=1126.440,-79.203,-46.778,179.510,4.813,148.963
C00700=1126.446,-79.453,-46.768,179.511,4.808,148.961
C00701=1126.451,-79.703,-46.759,179.511,4.803,148.960
C00702=1126.457,-79.952,-46.749,179.511,4.797,148.959
C00703=1126.462,-80.202,-46.740,179.511,4.792,148.958
C00704=1126.468,-80.452,-46.730,179.511,4.787,148.957
C00705=1126.473,-80.701,-46.721,179.511,4.782,148.956
C00706=1126.478,-80.951,-46.712,179.511,4.777,148.954
C00707=1126.484,-81.201,-46.702,179.512,4.772,148.953
C00708=1126.489,-81.451,-46.693,179.512,4.766,148.952
C00709=1126.494,-81.700,-46.684,179.512,4.761,148.951
C00710=1126.500,-81.951,-46.674,179.513,4.757,148.950
C00711=1126.505,-82.200,-46.665,179.513,4.752,148.949
C00712=1126.510,-82.450,-46.655,179.513,4.747,148.947
C00713=1126.516,-82.699,-46.647,179.513,4.741,148.946
C00714=1126.521,-82.949,-46.638,179.513,4.736,148.945
C00715=1126.527,-83.199,-46.628,179.514,4.731,148.944
C00716=1126.532,-83.448,-46.619,179.514,4.726,148.943
C00717=1126.537,-83.698,-46.610,179.514,4.721,148.942
C00718=1126.543,-83.948,-46.600,179.515,4.716,148.940
C00719=1126.548,-84.198,-46.591,179.515,4.711,148.939
C00720=1126.553,-84.448,-46.582,179.516,4.706,148.938
C00721=1126.558,-84.697,-46.573,179.516,4.701,148.937
C00722=1126.564,-84.948,-46.563,179.516,4.695,148.935
C00723=1126.569,-85.197,-46.554,179.517,4.691,148.934
C00724=1126.575,-85.447,-46.546,179.517,4.686,148.933
C00725=1126.580,-85.697,-46.536,179.517,4.681,148.932
C00726=1126.586,-85.947,-46.527,179.518,4.675,148.931
C00727=1126.591,-86.196,-46.518,179.518,4.671,148.929
C00728=1126.596,-86.446,-46.509,179.519,4.666,148.928
C00729=1126.602,-86.696,-46.500,179.519,4.660,148.927
C00730=1126.607,-86.946,-46.491,179.520,4.656,148.926
C00731=1126.612,-87.195,-46.482,179.520,4.651,148.925
C00732=1126.618,-87.445,-46.473,179.521,4.645,148.923
C00733=1126.624,-87.696,-46.463,179.521,4.641,148.922
C00734=1126.628,-87.911,-46.455,179.522,4.637,148.921
C00735=1126.633,-88.126,-46.448,179.522,4.633,148.920
C00736=1126.637,-88.342,-46.440,179.522,4.628,148.919
C00737=1126.641,-88.559,-46.433,179.523,4.624,148.918
C00738=1126.647,-88.774,-46.424,179.523,4.620,148.917
C00739=1126.651,-88.990,-46.416,179.524,4.615,148.916
C00740=1126.655,-89.206,-46.408,179.524,4.611,148.915
C00741=1126.660,-89.421,-46.401,179.525,4.607,148.914
C00742=1126.666,-89.671,-46.393,179.526,4.602,148.912
C00743=1126.671,-89.921,-46.382,179.526,4.597,148.911
C00744=1126.676,-90.171,-46.373,179.527,4.593,148.910
C00745=1126.682,-90.420,-46.365,179.527,4.587,148.909
C00746=1126.687,-90.670,-46.356,179.528,4.583,148.907
C00747=1126.692,-90.919,-46.347,179.528,4.578,148.906
C00748=1126.698,-91.170,-46.338,179.530,4.573,148.905
C00749=1126.704,-91.419,-46.329,179.530,4.568,148.904
C00750=1126.709,-91.669,-46.320,179.531,4.564,148.902
C00751=1126.714,-91.919,-46.311,179.531,4.559,148.901
C00752=1126.720,-92.168,-46.302,179.532,4.554,148.900
C00753=1126.725,-92.418,-46.294,179.533,4.549,148.899
C00754=1126.730,-92.668,-46.285,179.534,4.545,148.897
C00755=1126.736,-92.918,-46.275,179.534,4.539,148.896
C00756=1126.741,-93.168,-46.266,179.535,4.535,148.895
C00757=1126.746,-93.418,-46.257,179.536,4.531,148.894
C00758=1126.752,-93.668,-46.250,179.536,4.526,148.892
C00759=1126.757,-93.918,-46.241,179.537,4.521,148.891
C00760=1126.763,-94.167,-46.232,179.538,4.516,148.890
C00761=1126.768,-94.417,-46.223,179.539,4.512,148.889
C00762=1126.774,-94.667,-46.213,179.539,4.507,148.888
C00763=1126.779,-94.917,-46.205,179.539,4.502,148.886
C00764=1126.785,-95.166,-46.196,179.540,4.497,148.885
C00765=1126.790,-95.416,-46.187,179.540,4.492,148.884
C00766=1126.795,-95.666,-46.178,179.541,4.487,148.883
C00767=1126.801,-95.915,-46.170,179.541,4.482,148.882
C00768=1126.806,-96.165,-46.161,179.542,4.478,148.880
C00769=1126.811,-96.415,-46.152,179.542,4.472,148.879
C00770=1126.817,-96.665,-46.144,179.542,4.467,148.878
C00771=1126.822,-96.915,-46.135,179.542,4.462,148.877
C00772=1126.827,-97.164,-46.126,179.542,4.457,148.876
C00773=1126.833,-97.414,-46.117,179.543,4.453,148.875
C00774=1126.838,-97.664,-46.108,179.543,4.448,148.874
C00775=1126.844,-97.914,-46.099,179.543,4.443,148.872
C00776=1126.850,-98.164,-46.091,179.543,4.437,148.871
C00777=1126.855,-98.414,-46.082,179.544,4.432,148.870
C00778=1126.860,-98.664,-46.073,179.544,4.427,148.869
C00779=1126.866,-98.913,-46.065,179.545,4.423,148.868
C00780=1126.871,-99.163,-46.056,179.545,4.417,148.866
C00781=1126.877,-99.413,-46.048,179.545,4.413,148.865
C00782=1126.882,-99.663,-46.039,179.545,4.408,148.864
C00783=1126.887,-99.912,-46.030,179.545,4.402,148.863
C00784=1126.893,-100.162,-46.021,179.545,4.397,148.862
C00785=1126.898,-100.412,-46.012,179.546,4.393,148.861
C00786=1126.904,-100.662,-46.005,179.546,4.388,148.860
C00787=1126.909,-100.912,-45.996,179.546,4.382,148.858
C00788=1126.914,-101.161,-45.987,179.547,4.377,148.857
C00789=1126.920,-101.411,-45.979,179.546,4.373,148.856
C00790=1126.928,-101.779,-45.966,179.547,4.365,148.854
C00791=1126.953,-102.989,-45.921,178.577,6.164,149.532
C00792=1126.959,-103.262,-45.912,178.574,6.163,149.532
C00793=1126.965,-103.535,-45.902,178.572,6.162,149.533
C00794=1126.970,-103.807,-45.893,178.571,6.162,149.533
C00795=1126.977,-104.057,-45.883,178.568,6.162,149.534
C00796=1126.982,-104.306,-45.875,178.566,6.161,149.534
C00797=1126.987,-104.556,-45.866,178.565,6.161,149.535
C00798=1126.992,-104.806,-45.857,178.562,6.160,149.535
C00799=1126.998,-105.056,-45.848,178.561,6.160,149.536
C00800=1127.003,-105.305,-45.839,178.559,6.159,149.536
C00801=1127.009,-105.555,-45.830,178.556,6.159,149.537
C00802=1127.014,-105.805,-45.821,178.555,6.159,149.537
C00803=1127.019,-106.055,-45.813,178.553,6.158,149.538
C00804=1127.025,-106.304,-45.805,178.550,6.157,149.538
C00805=1127.030,-106.554,-45.796,178.549,6.157,149.538
C00806=1127.035,-106.804,-45.787,178.547,6.157,149.539
C00807=1127.040,-107.054,-45.778,178.545,6.157,149.539
C00808=1127.046,-107.304,-45.769,178.543,6.156,149.540
C00809=1127.051,-107.553,-45.761,178.541,6.155,149.540
C00810=1127.057,-107.803,-45.752,178.540,6.155,149.541
C00811=1127.062,-108.053,-45.744,178.537,6.154,149.541
C00812=1127.067,-108.303,-45.735,178.535,6.153,149.542
C00813=1127.073,-108.552,-45.726,178.534,6.153,149.542
C00814=1127.078,-108.802,-45.717,178.531,6.153,149.543
C00815=1127.083,-109.052,-45.708,178.530,6.153,149.543
C00816=1127.089,-109.302,-45.701,178.528,6.152,149.544
C00817=1127.094,-109.552,-45.692,178.525,6.151,149.544
C00818=1127.100,-109.802,-45.683,178.524,6.151,149.545
C00819=1127.105,-110.051,-45.674,178.522,6.150,149.545
C00820=1127.111,-110.301,-45.665,178.520,6.151,149.546
C00821=1127.116,-110.551,-45.657,178.518,6.150,149.546
C00822=1127.121,-110.801,-45.648,178.516,6.149,149.547
C00823=1127.126,-111.051,-45.639,178.514,6.149,149.547
C00824=1127.132,-111.300,-45.631,178.512,6.148,149.548
C00825=1127.138,-111.550,-45.623,178.510,6.148,149.548
C00826=1127.143,-111.800,-45.614,178.508,6.148,149.548
C00827=1127.149,-112.049,-45.605,178.506,6.147,149.549
C00828=1127.154,-112.300,-45.597,178.505,6.147,149.549
C00829=1127.159,-112.550,-45.588,178.502,6.146,149.550
C00830=1127.165,-112.799,-45.580,178.501,6.146,149.550
C00831=1127.170,-113.049,-45.571,178.499,6.145,149.551
C00832=1127.176,-113.299,-45.562,178.496,6.144,149.551
C00833=1127.181,-113.548,-45.554,178.495,6.144,149.552
C00834=1127.187,-113.798,-45.545,178.493,6.144,149.552
C00835=1127.192,-114.049,-45.537,178.491,6.144,149.553
C00836=1127.197,-114.298,-45.528,178.489,6.143,149.553
C00837=1127.202,-114.547,-45.520,178.487,6.143,149.554
C00838=1127.208,-114.798,-45.512,178.485,6.142,149.554
C00839=1127.213,-115.047,-45.503,178.483,6.142,149.555
C00840=1127.219,-115.297,-45.494,178.482,6.141,149.555
C00841=1127.224,-115.547,-45.486,178.480,6.140,149.555
C00842=1127.230,-115.796,-45.478,178.478,6.141,149.556
C00843=1127.235,-116.046,-45.469,178.476,6.140,149.556
C00844=1127.240,-116.297,-45.461,178.474,6.139,149.557
C00845=1127.246,-116.546,-45.452,178.472,6.139,149.557
C00846=1127.251,-116.796,-45.445,178.470,6.138,149.558
C00847=1127.256,-117.046,-45.436,178.468,6.138,149.558
C00848=1127.262,-117.295,-45.427,178.466,6.138,149.559
C00849=1127.267,-117.545,-45.419,178.464,6.138,149.559
C00850=1127.273,-117.795,-45.410,178.462,6.137,149.560
C00851=1127.279,-118.045,-45.402,178.460,6.136,149.560
C00852=1127.284,-118.295,-45.393,178.459,6.136,149.560
C00853=1127.289,-118.544,-45.386,178.457,6.135,149.561
C00854=1127.294,-118.794,-45.377,178.455,6.135,149.561
C00855=1127.299,-119.044,-45.368,178.453,6.134,149.562
C00856=1127.306,-119.294,-45.360,178.451,6.135,149.562
C00857=1127.311,-119.544,-45.352,178.449,6.134,149.563
C00858=1127.316,-119.793,-45.344,178.448,6.134,149.563
C00859=1127.321,-120.043,-45.335,178.445,6.133,149.564
C00860=1127.327,-120.294,-45.327,178.444,6.132,149.564
C00861=1127.332,-120.543,-45.319,178.442,6.132,149.565
C00862=1127.338,-120.793,-45.311,178.440,6.131,149.565
C00863=1127.343,-121.042,-45.303,178.438,6.131,149.566
C00864=1127.348,-121.292,-45.294,178.436,6.131,149.566
C00865=1127.354,-121.542,-45.286,178.434,6.131,149.567
C00866=1127.360,-121.792,-45.278,178.432,6.130,149.567
C00867=1127.365,-122.042,-45.269,178.431,6.130,149.568
C00868=1127.370,-122.291,-45.262,178.429,6.129,149.568
C00869=1127.375,-122.541,-45.253,178.427,6.129,149.568
C00870=1127.381,-122.791,-45.245,178.425,6.128,149.569
C00871=1127.387,-123.041,-45.236,178.423,6.127,149.569
C00872=1127.391,-123.291,-45.228,178.421,6.127,149.570
C00873=1127.397,-123.541,-45.221,178.419,6.127,149.570
C00874=1127.403,-123.791,-45.212,178.418,6.127,149.571
C00875=1127.409,-124.040,-45.204,178.415,6.126,149.571
C00876=1127.413,-124.290,-45.196,178.414,6.126,149.572
C00877=1127.419,-124.540,-45.188,178.412,6.125,149.572
C00878=1127.424,-124.790,-45.179,178.410,6.125,149.572
C00879=1127.430,-125.039,-45.172,178.408,6.124,149.573
C00880=1127.435,-125.289,-45.163,178.407,6.124,149.573
C00881=1127.440,-125.539,-45.155,178.404,6.124,149.574
C00882=1127.446,-125.789,-45.147,178.403,6.124,149.574
C00883=1127.451,-126.039,-45.138,178.401,6.123,149.575
C00884=1127.457,-126.288,-45.131,178.399,6.123,149.575
C00885=1127.462,-126.539,-45.122,178.397,6.122,149.576
C00886=1127.467,-126.788,-45.114,178.396,6.122,149.576
C00887=1127.473,-127.038,-45.106,178.393,6.121,149.577
C00888=1127.479,-127.288,-45.098,178.391,6.120,149.577
C00889=1127.483,-127.537,-45.090,178.390,6.120,149.577
C00890=1127.489,-127.787,-45.082,178.388,6.119,149.578
C00891=1127.495,-128.038,-45.074,178.386,6.119,149.578
C00892=1127.500,-128.287,-45.066,178.384,6.119,149.579
C00893=1127.505,-128.537,-45.058,178.383,6.119,149.579
C00894=1127.511,-128.787,-45.050,178.380,6.118,149.580
C00895=1127.090,-128.798,-45.094,178.378,6.122,149.581
C00896=1127.084,-128.548,-45.102,178.380,6.122,149.581
C00897=1127.079,-128.298,-45.111,178.381,6.123,149.581
C00898=1127.074,-128.049,-45.118,178.383,6.123,149.580
C00899=1127.068,-127.798,-45.126,178.385,6.123,149.580
C00900=1127.063,-127.549,-45.135,178.387,6.124,149.579
C00901=1127.058,-127.299,-45.143,178.389,6.124,149.579
C00902=1127.052,-127.049,-45.151,178.391,6.125,149.578
C00903=1127.047,-126.799,-45.159,178.392,6.125,149.578
C00904=1127.042,-126.549,-45.167,178.394,6.126,149.577
C00905=1127.036,-126.300,-45.175,178.396,6.126,149.577
C00906=1127.031,-126.050,-45.184,178.398,6.127,149.577
C00907=1127.025,-125.800,-45.191,178.399,6.127,149.576
C00908=1127.020,-125.550,-45.200,178.402,6.127,149.576
C00909=1127.014,-125.301,-45.208,178.403,6.127,149.575
C00910=1127.009,-125.050,-45.216,178.405,6.128,149.575
C00911=1127.004,-124.801,-45.224,178.407,6.128,149.574
C00912=1126.998,-124.551,-45.232,178.409,6.129,149.574
C00913=1126.992,-124.302,-45.240,178.410,6.129,149.573
C00914=1126.987,-124.051,-45.249,178.413,6.130,149.573
C00915=1126.982,-123.802,-45.257,178.414,6.130,149.572
C00916=1126.976,-123.552,-45.265,178.416,6.130,149.572
C00917=1126.971,-123.301,-45.273,178.418,6.132,149.572
C00918=1126.966,-123.053,-45.281,178.420,6.131,149.571
C00919=1126.960,-122.802,-45.289,178.422,6.132,149.571
C00920=1126.955,-122.553,-45.298,178.423,6.132,149.570
C00921=1126.949,-122.302,-45.306,178.426,6.133,149.570
C00922=1126.944,-122.054,-45.314,178.427,6.133,149.569
C00923=1126.939,-121.803,-45.322,178.429,6.134,149.569
C00924=1126.933,-121.553,-45.331,178.431,6.134,149.568
C00925=1126.927,-121.304,-45.339,178.433,6.135,149.568
C00926=1126.922,-121.054,-45.347,178.434,6.135,149.567
C00927=1126.917,-120.804,-45.355,178.437,6.135,149.567
C00928=1126.912,-120.554,-45.364,178.439,6.136,149.566
C00929=1126.906,-120.304,-45.372,178.440,6.136,149.566
C00930=1126.900,-120.055,-45.380,178.443,6.137,149.565
C00931=1126.895,-119.804,-45.388,178.444,6.137,149.565
C00932=1126.890,-119.555,-45.396,178.446,6.138,149.565
C00933=1126.884,-119.305,-45.405,178.447,6.138,149.564
C00934=1126.879,-119.055,-45.413,178.450,6.139,149.564
C00935=1126.873,-118.805,-45.421,178.451,6.139,149.563
C00936=1126.868,-118.556,-45.430,178.453,6.139,149.563
C00937=1126.863,-118.307,-45.438,178.456,6.140,149.562
C00938=1126.858,-118.056,-45.446,178.457,6.140,149.562
C00939=1126.852,-117.806,-45.455,178.459,6.141,149.561
C00940=1126.846,-117.557,-45.463,178.461,6.141,149.561
C00941=1126.841,-117.307,-45.472,178.463,6.142,149.561
C00942=1126.835,-117.057,-45.480,178.464,6.142,149.560
C00943=1126.830,-116.807,-45.489,178.467,6.142,149.560
C00944=1126.825,-116.558,-45.497,178.469,6.143,149.559
C00945=1126.819,-116.308,-45.505,178.470,6.143,149.559
C00946=1126.814,-116.058,-45.514,178.473,6.144,149.558
C00947=1126.809,-115.807,-45.522,178.474,6.144,149.558
C00948=1126.803,-115.558,-45.530,178.476,6.145,149.557
C00949=1126.798,-115.308,-45.539,178.478,6.145,149.557
C00950=1126.792,-115.058,-45.547,178.480,6.145,149.556
C00951=1126.787,-114.809,-45.556,178.482,6.146,149.556
C00952=1126.782,-114.559,-45.564,178.483,6.146,149.555
C00953=1126.777,-114.309,-45.572,178.486,6.147,149.555
C00954=1126.771,-114.060,-45.581,178.487,6.147,149.554
C00955=1126.766,-113.810,-45.590,178.489,6.148,149.554
C00956=1126.760,-113.559,-45.598,178.491,6.148,149.553
C00957=1126.755,-113.310,-45.607,178.493,6.148,149.553
C00958=1126.749,-113.060,-45.616,178.495,6.149,149.552
C00959=1126.744,-112.810,-45.624,178.497,6.149,149.552
C00960=1126.739,-112.583,-45.632,178.499,6.150,149.552
C00961=1126.734,-112.357,-45.639,178.500,6.150,149.551
C00962=1126.729,-112.131,-45.647,178.503,6.151,149.551
C00963=1126.705,-111.004,-45.686,179.561,4.179,148.810
C00964=1126.700,-110.754,-45.695,179.561,4.184,148.811
C00965=1126.694,-110.504,-45.702,179.561,4.190,148.812
C00966=1126.689,-110.254,-45.711,179.560,4.195,148.813
C00967=1126.683,-110.005,-45.719,179.561,4.201,148.815
C00968=1126.678,-109.755,-45.727,179.560,4.206,148.816
C00969=1126.672,-109.505,-45.735,179.560,4.211,148.817
C00970=1126.667,-109.255,-45.744,179.560,4.216,148.818
C00971=1126.661,-109.006,-45.751,179.560,4.221,148.819
C00972=1126.656,-108.756,-45.760,179.559,4.227,148.821
C00973=1126.651,-108.505,-45.768,179.559,4.232,148.822
C00974=1126.645,-108.256,-45.777,179.559,4.237,148.823
C00975=1126.640,-108.006,-45.785,179.559,4.242,148.824
C00976=1126.635,-107.757,-45.793,179.559,4.247,148.825
C00977=1126.629,-107.507,-45.801,179.559,4.252,148.826
C00978=1126.624,-107.257,-45.810,179.558,4.257,148.828
C00979=1126.618,-107.007,-45.818,179.558,4.262,148.829
C00980=1126.613,-106.757,-45.827,179.558,4.268,148.830
C00981=1126.607,-106.508,-45.835,179.558,4.273,148.831
C00982=1126.601,-106.257,-45.844,179.558,4.278,148.832
C00983=1126.597,-106.008,-45.852,179.557,4.283,148.834
C00984=1126.591,-105.758,-45.860,179.558,4.288,148.834
C00985=1126.586,-105.508,-45.869,179.557,4.293,148.836
C00986=1126.581,-105.258,-45.878,179.557,4.298,148.837
C00987=1126.575,-105.009,-45.885,179.557,4.303,148.838
C00988=1126.569,-104.759,-45.894,179.557,4.309,148.839
C00989=1126.564,-104.508,-45.902,179.556,4.313,148.840
C00990=1126.558,-104.259,-45.911,179.556,4.318,148.842
C00991=1126.554,-104.010,-45.919,179.555,4.323,148.843
C00992=1126.548,-103.759,-45.927,179.555,4.329,148.844
C00993=1126.542,-103.510,-45.936,179.555,4.333,148.845
C00994=1126.537,-103.260,-45.945,179.555,4.338,148.846
C00995=1126.532,-103.010,-45.953,179.555,4.344,148.847
C00996=1126.523,-102.608,-45.967,179.554,4.352,148.849
C00997=1126.515,-102.206,-45.981,179.554,4.360,148.851
C00998=1126.506,-101.804,-45.995,179.554,4.368,148.853
C00999=1126.497,-101.402,-46.008,179.553,4.376,148.855
C01000=1126.492,-101.153,-46.017,179.553,4.381,148.856
C01001=1126.486,-100.903,-46.026,179.553,4.386,148.857
C01002=1126.481,-100.652,-46.034,179.553,4.391,148.858
C01003=1126.475,-100.403,-46.042,179.553,4.397,148.859
C01004=1126.470,-100.153,-46.051,179.552,4.401,148.861
C01005=1126.465,-99.904,-46.060,179.552,4.406,148.862
C01006=1126.459,-99.653,-46.068,179.551,4.411,148.863
C01007=1126.454,-99.404,-46.077,179.551,4.416,148.864
C01008=1126.448,-99.154,-46.086,179.551,4.422,148.865
C01009=1126.443,-98.904,-46.095,179.551,4.427,148.867
C01010=1126.437,-98.654,-46.104,179.551,4.431,148.868
C01011=1126.432,-98.405,-46.113,179.550,4.436,148.869
C01012=1126.426,-98.154,-46.121,179.550,4.441,148.870
C01013=1126.421,-97.905,-46.130,179.550,4.446,148.871
C01014=1126.416,-97.655,-46.139,179.550,4.451,148.872
C01015=1126.410,-97.406,-46.147,179.549,4.457,148.873
C01016=1126.405,-97.156,-46.156,179.549,4.461,148.875
C01017=1126.400,-96.906,-46.165,179.548,4.466,148.876
C01018=1126.395,-96.656,-46.174,179.548,4.471,148.877
C01019=1126.388,-96.406,-46.182,179.548,4.476,148.878
C01020=1126.383,-96.156,-46.191,179.548,4.481,148.879
C01021=1126.378,-95.907,-46.200,179.548,4.486,148.880
C01022=1126.373,-95.657,-46.208,179.547,4.491,148.882
C01023=1126.366,-95.407,-46.218,179.547,4.496,148.883
C01024=1126.361,-95.157,-46.227,179.547,4.501,148.884
C01025=1126.356,-94.908,-46.235,179.546,4.505,148.885
C01026=1126.351,-94.658,-46.244,179.546,4.511,148.886
C01027=1126.346,-94.408,-46.253,179.546,4.516,148.887
C01028=1126.340,-94.159,-46.262,179.545,4.520,148.889
C01029=1126.335,-93.909,-46.271,179.544,4.525,148.890
C01030=1126.330,-93.659,-46.280,179.543,4.529,148.891
C01031=1126.324,-93.409,-46.289,179.543,4.534,148.892
C01032=1126.319,-93.159,-46.298,179.542,4.539,148.894
C01033=1126.313,-92.909,-46.307,179.541,4.544,148.895
C01034=1126.308,-92.660,-46.315,179.540,4.549,148.896
C01035=1126.302,-92.410,-46.324,179.540,4.553,148.897
C01036=1126.297,-92.160,-46.333,179.539,4.557,148.899
C01037=1126.291,-91.910,-46.343,179.538,4.563,148.900
C01038=1126.286,-91.660,-46.352,179.537,4.567,148.901
C01039=1126.281,-91.410,-46.360,179.536,4.572,148.902
C01040=1126.275,-91.161,-46.369,179.536,4.577,148.904
C01041=1126.270,-90.911,-46.378,179.535,4.582,148.905
C01042=1126.264,-90.661,-46.387,179.535,4.587,148.906
C01043=1126.259,-90.411,-46.396,179.534,4.591,148.907
C01044=1126.254,-90.162,-46.405,179.533,4.597,148.909
C01045=1126.249,-89.912,-46.414,179.533,4.601,148.910
C01046=1126.244,-89.662,-46.423,179.532,4.606,148.911
C01047=1126.237,-89.412,-46.432,179.532,4.611,148.912
C01048=1126.233,-89.197,-46.440,179.531,4.615,148.913
C01049=1126.229,-88.981,-46.448,179.530,4.619,148.914
C01050=1126.224,-88.766,-46.456,179.530,4.623,148.916
C01051=1126.219,-88.549,-46.463,179.529,4.627,148.917
C01052=1126.214,-88.333,-46.471,179.529,4.632,148.918
C01053=1126.210,-88.118,-46.479,179.529,4.636,148.919
C01054=1126.205,-87.902,-46.487,179.528,4.641,148.920
C01055=1126.201,-87.686,-46.495,179.528,4.645,148.921
C01056=1126.195,-87.436,-46.505,179.528,4.650,148.922
C01057=1126.190,-87.186,-46.513,179.526,4.655,148.923
C01058=1126.184,-86.937,-46.522,179.526,4.660,148.925
C01059=1126.179,-86.687,-46.531,179.526,4.665,148.926
C01060=1126.173,-86.437,-46.540,179.525,4.669,148.927
C01061=1126.168,-86.188,-46.550,179.525,4.674,148.928
C01062=1126.163,-85.938,-46.559,179.524,4.680,148.929
C01063=1126.158,-85.688,-46.568,179.524,4.684,148.931
C01064=1126.152,-85.438,-46.577,179.524,4.690,148.932
C01065=1126.147,-85.188,-46.586,179.523,4.695,148.933
C01066=1126.142,-84.939,-46.596,179.523,4.700,148.934
C01067=1126.136,-84.689,-46.605,179.522,4.704,148.935
C01068=1126.131,-84.439,-46.614,179.522,4.709,148.937
C01069=1126.126,-84.189,-46.623,179.522,4.715,148.938
C01070=1126.120,-83.939,-46.633,179.521,4.720,148.939
C01071=1126.115,-83.690,-46.642,179.521,4.725,148.940
C01072=1126.110,-83.440,-46.651,179.520,4.730,148.941
C01073=1126.104,-83.190,-46.661,179.520,4.735,148.943
C01074=1126.098,-82.941,-46.669,179.520,4.740,148.944
C01075=1126.093,-82.691,-46.679,179.520,4.745,148.945
C01076=1126.087,-82.441,-46.688,179.520,4.750,148.946
C01077=1126.082,-82.191,-46.697,179.520,4.755,148.947
C01078=1126.077,-81.942,-46.707,179.519,4.761,148.948
C01079=1126.072,-81.692,-46.716,179.519,4.766,148.950
C01080=1126.066,-81.442,-46.725,179.519,4.771,148.951
C01081=1126.061,-81.193,-46.735,179.518,4.776,148.952
C01082=1126.056,-80.943,-46.744,179.518,4.781,148.953
C01083=1126.050,-80.693,-46.753,179.517,4.786,148.955
C01084=1126.045,-80.443,-46.763,179.517,4.791,148.956
C01085=1126.040,-80.193,-46.772,179.517,4.796,148.957
C01086=1126.034,-79.943,-46.782,179.517,4.801,148.958
C01087=1126.029,-79.694,-46.791,179.517,4.807,148.959
C01088=1126.023,-79.444,-46.801,179.517,4.813,148.960
C01089=1126.018,-79.194,-46.810,179.517,4.818,148.962
C01090=1126.013,-78.945,-46.819,179.517,4.823,148.962
C01091=1126.007,-78.695,-46.829,179.517,4.828,148.964
C01092=1126.002,-78.445,-46.838,179.517,4.833,148.965
C01093=1125.996,-78.195,-46.848,179.517,4.838,148.966
C01094=1125.992,-77.945,-46.857,179.517,4.843,148.967
C01095=1125.986,-77.695,-46.867,179.517,4.848,148.968
C01096=1125.981,-77.445,-46.876,179.517,4.854,148.969
C01097=1125.975,-77.196,-46.887,179.516,4.859,148.971
C01098=1125.970,-76.946,-46.895,179.516,4.864,148.972
C01099=1125.965,-76.696,-46.906,179.517,4.870,148.973
C01100=1125.959,-76.447,-46.915,179.517,4.875,148.974
C01101=1125.954,-76.197,-46.925,179.517,4.880,148.975
C01102=1125.949,-75.947,-46.934,179.517,4.885,148.976
C01103=1125.943,-75.698,-46.944,179.517,4.890,148.977
C01104=1125.939,-75.482,-46.952,179.517,4.895,148.978
C01105=1125.934,-75.266,-46.960,179.517,4.900,148.979
C01106=1125.929,-75.051,-46.968,179.517,4.904,148.980
C01107=1125.924,-74.835,-46.977,179.517,4.908,148.981
C01108=1125.920,-74.619,-46.985,179.517,4.913,148.982
C01109=1125.915,-74.403,-46.994,179.517,4.917,148.983
C01110=1125.911,-74.187,-47.002,179.517,4.922,148.984
C01111=1125.906,-73.972,-47.010,179.518,4.927,148.985
C01112=1125.901,-73.723,-47.020,179.518,4.932,148.986
C01113=1125.896,-73.472,-47.030,179.518,4.937,148.987
C01114=1125.890,-73.222,-47.040,179.518,4.943,148.988
C01115=1125.885,-72.973,-47.049,179.518,4.948,148.989
C01116=1125.879,-72.723,-47.059,179.519,4.953,148.990
C01117=1125.874,-72.474,-47.068,179.519,4.959,148.992
C01118=1125.869,-72.224,-47.079,179.519,4.964,148.993
C01119=1125.863,-71.974,-47.088,179.519,4.969,148.994
C01120=1125.858,-71.724,-47.098,179.520,4.975,148.995
C01121=1125.853,-71.475,-47.108,179.520,4.979,148.996
C01122=1125.847,-71.224,-47.118,179.520,4.985,148.997
C01123=1125.842,-70.975,-47.127,179.520,4.991,148.998
C01124=1125.836,-70.726,-47.138,179.521,4.995,148.999
C01125=1125.831,-70.476,-47.148,179.521,5.001,149.000
C01126=1125.826,-70.225,-47.157,179.522,5.006,149.001
C01127=1125.821,-69.976,-47.167,179.522,5.012,149.002
C01128=1125.815,-69.726,-47.178,179.522,5.017,149.003
C01129=1125.810,-69.477,-47.186,179.522,5.022,149.004
C01130=1125.804,-69.227,-47.197,179.523,5.028,149.005
C01131=1125.799,-68.977,-47.207,179.523,5.033,149.006
C01132=1125.794,-68.727,-47.217,179.524,5.038,149.007
C01133=1125.789,-68.478,-47.227,179.524,5.043,149.008
C01134=1125.783,-68.228,-47.237,179.525,5.049,149.009
C01135=1125.778,-67.978,-47.247,179.525,5.054,149.010
C01136=1125.772,-67.728,-47.257,179.526,5.060,149.011
C01137=1125.767,-67.479,-47.267,179.526,5.064,149.012
C01138=1125.762,-67.229,-47.277,179.527,5.070,149.013
C01139=1125.757,-66.979,-47.288,179.528,5.076,149.014
C01140=1125.751,-66.729,-47.297,179.528,5.081,149.015
C01141=1125.746,-66.480,-47.307,179.529,5.086,149.016
C01142=1125.741,-66.230,-47.317,179.529,5.091,149.017
C01143=1125.736,-65.980,-47.328,179.530,5.097,149.018
C01144=1125.730,-65.730,-47.338,179.530,5.102,149.019
C01145=1125.724,-65.481,-47.348,179.531,5.107,149.020
C01146=1125.719,-65.231,-47.358,179.532,5.113,149.021
C01147=1125.714,-64.981,-47.368,179.533,5.118,149.022
C01148=1125.709,-64.732,-47.378,179.533,5.124,149.023
C01149=1125.703,-64.482,-47.389,179.533,5.128,149.024
C01150=1125.698,-64.232,-47.399,179.534,5.134,149.025
C01151=1125.693,-63.982,-47.409,179.535,5.140,149.026
C01152=1125.687,-63.733,-47.420,179.536,5.144,149.027
C01153=1125.683,-63.483,-47.430,179.537,5.150,149.028
C01154=1125.677,-63.233,-47.440,179.538,5.155,149.029
C01155=1125.672,-62.984,-47.450,179.538,5.160,149.029
C01156=1125.667,-62.734,-47.461,179.539,5.166,149.030
C01157=1125.661,-62.484,-47.471,179.540,5.171,149.031
C01158=1125.655,-62.235,-47.481,179.540,5.176,149.032
C01159=1125.650,-61.984,-47.492,179.541,5.182,149.033
C01160=1125.646,-61.769,-47.501,179.542,5.186,149.034
C01161=1125.642,-61.554,-47.510,179.543,5.191,149.035
C01162=1125.637,-61.337,-47.518,179.544,5.195,149.035
C01163=1125.632,-61.122,-47.527,179.545,5.201,149.036
C01164=1125.628,-60.906,-47.537,179.545,5.205,149.037
C01165=1125.623,-60.691,-47.546,179.546,5.209,149.038
C01166=1125.619,-60.475,-47.554,179.547,5.214,149.039
C01167=1125.614,-60.260,-47.563,179.548,5.219,149.039
C01168=1125.609,-60.010,-47.573,179.547,5.223,149.040
C01169=1125.604,-59.761,-47.585,179.547,5.228,149.041
C01170=1125.598,-59.511,-47.595,179.547,5.233,149.042
C01171=1125.593,-59.261,-47.606,179.547,5.237,149.043
C01172=1125.588,-59.011,-47.616,179.547,5.242,149.045
C01173=1125.582,-58.762,-47.626,179.546,5.246,149.046
C01174=1125.577,-58.512,-47.637,179.547,5.251,149.047
C01175=1125.572,-58.262,-47.647,179.546,5.255,149.048
C01176=1125.567,-58.012,-47.658,179.546,5.261,149.049
C01177=1125.561,-57.763,-47.668,179.546,5.265,149.050
C01178=1125.556,-57.512,-47.679,179.546,5.270,149.051
C01179=1125.551,-57.264,-47.690,179.545,5.274,149.052
C01180=1125.546,-57.013,-47.700,179.545,5.279,149.053
C01181=1125.540,-56.764,-47.711,179.545,5.284,149.054
C01182=1125.535,-56.514,-47.722,179.545,5.288,149.055
C01183=1125.529,-56.264,-47.733,179.545,5.293,149.056
C01184=1125.524,-56.015,-47.743,179.544,5.297,149.057
C01185=1125.519,-55.764,-47.753,179.545,5.302,149.058
C01186=1125.513,-55.516,-47.764,179.544,5.307,149.059
C01187=1125.508,-55.265,-47.775,179.544,5.312,149.061
C01188=1125.503,-55.016,-47.785,179.544,5.316,149.062
C01189=1125.498,-54.766,-47.796,179.543,5.321,149.063
C01190=1125.492,-54.517,-47.807,179.543,5.326,149.064
C01191=1125.487,-54.266,-47.817,179.543,5.330,149.065
C01192=1125.482,-54.017,-47.828,179.543,5.335,149.066
C01193=1125.476,-53.767,-47.839,179.542,5.339,149.067
C01194=1125.471,-53.517,-47.850,179.542,5.344,149.068
C01195=1125.466,-53.268,-47.861,179.542,5.348,149.069
C01196=1125.461,-53.018,-47.871,179.542,5.354,149.070
C01197=1125.456,-52.769,-47.882,179.542,5.359,149.071
C01198=1125.450,-52.519,-47.893,179.542,5.363,149.072
C01199=1125.445,-52.269,-47.903,179.542,5.368,149.073
C01200=1125.440,-52.019,-47.915,179.541,5.372,149.075
C01201=1125.434,-51.769,-47.925,179.541,5.377,149.076
C01202=1125.430,-51.520,-47.936,179.541,5.381,149.077
C01203=1125.424,-51.270,-47.947,179.541,5.386,149.078
C01204=1125.419,-51.020,-47.957,179.541,5.391,149.079
C01205=1125.414,-50.771,-47.968,179.540,5.396,149.080
C01206=1125.408,-50.520,-47.979,179.540,5.401,149.081
C01207=1125.403,-50.271,-47.990,179.540,5.405,149.082
C01208=1125.398,-50.021,-48.001,179.540,5.410,149.083
C01209=1125.392,-49.772,-48.012,179.539,5.414,149.084
C01210=1125.387,-49.522,-48.022,179.539,5.419,149.085
C01211=1125.382,-49.272,-48.034,179.540,5.424,149.086
C01212=1125.376,-49.023,-48.044,179.539,5.428,149.087
C01213=1125.372,-48.773,-48.056,179.539,5.433,149.089
C01214=1125.366,-48.523,-48.066,179.538,5.438,149.090
C01215=1125.361,-48.273,-48.078,179.539,5.443,149.091
C01216=1125.356,-48.058,-48.087,179.539,5.447,149.092
C01217=1125.351,-47.842,-48.096,179.538,5.451,149.092
C01218=1125.347,-47.627,-48.106,179.538,5.454,149.093
C01219=1125.342,-47.411,-48.115,179.538,5.459,149.094
C01220=1125.337,-47.196,-48.124,179.537,5.463,149.095
C01221=1125.334,-46.980,-48.135,179.537,5.467,149.096
C01222=1125.329,-46.765,-48.144,179.537,5.471,149.097
C01223=1125.324,-46.549,-48.153,179.537,5.475,149.098
C01224=1125.319,-46.301,-48.164,179.537,5.480,149.099
C01225=1125.313,-46.050,-48.175,179.537,5.485,149.100
C01226=1125.309,-45.800,-48.187,179.537,5.489,149.101
C01227=1125.303,-45.551,-48.197,179.536,5.494,149.102
C01228=1125.298,-45.301,-48.208,179.537,5.499,149.103
C01229=1125.293,-45.051,-48.220,179.536,5.503,149.105
C01230=1125.287,-44.802,-48.230,179.536,5.508,149.106
C01231=1125.283,-44.552,-48.241,179.536,5.513,149.107
C01232=1125.276,-44.302,-48.252,179.536,5.517,149.108
C01233=1125.272,-44.053,-48.264,179.535,5.522,149.109
C01234=1125.267,-43.803,-48.275,179.535,5.527,149.110
C01235=1125.261,-43.553,-48.286,179.535,5.532,149.111
C01236=1125.256,-43.303,-48.297,179.535,5.536,149.112
C01237=1125.251,-43.054,-48.308,179.535,5.541,149.113
C01238=1125.245,-42.804,-48.319,179.537,5.547,149.114
C01239=1125.240,-42.554,-48.330,179.539,5.553,149.114
C01240=1125.235,-42.304,-48.342,179.541,5.559,149.115
C01241=1125.229,-42.055,-48.353,179.542,5.564,149.116
C01242=1125.224,-41.805,-48.364,179.544,5.570,149.117
C01243=1125.219,-41.555,-48.376,179.546,5.576,149.117
C01244=1125.214,-41.306,-48.387,179.548,5.582,149.118
C01245=1125.208,-41.056,-48.398,179.549,5.587,149.119
C01246=1125.203,-40.806,-48.409,179.551,5.592,149.120
C01247=1125.198,-40.556,-48.421,179.553,5.598,149.120
C01248=1125.193,-40.307,-48.432,179.554,5.603,149.121
C01249=1125.188,-40.058,-48.443,179.555,5.609,149.122
C01250=1125.182,-39.808,-48.455,179.557,5.614,149.122
C01251=1125.178,-39.558,-48.466,179.559,5.619,149.123
C01252=1125.172,-39.309,-48.478,179.560,5.625,149.124
C01253=1125.166,-39.058,-48.489,179.561,5.630,149.125
C01254=1125.161,-38.809,-48.500,179.563,5.635,149.125
C01255=1125.156,-38.559,-48.512,179.563,5.640,149.126
C01256=1125.151,-38.310,-48.523,179.565,5.645,149.127
C01257=1125.145,-38.060,-48.535,179.566,5.650,149.128
C01258=1125.140,-37.810,-48.546,179.567,5.656,149.128
C01259=1125.135,-37.560,-48.558,179.568,5.660,149.129
C01260=1125.130,-37.311,-48.569,179.569,5.666,149.130
C01261=1125.124,-37.062,-48.581,179.570,5.670,149.131
C01262=1125.119,-36.812,-48.593,179.571,5.676,149.132
C01263=1125.114,-36.562,-48.604,179.572,5.680,149.132
C01264=1125.109,-36.312,-48.616,179.573,5.685,149.133
C01265=1125.104,-36.062,-48.627,179.573,5.689,149.134
C01266=1125.099,-35.812,-48.639,179.575,5.695,149.135
C01267=1125.093,-35.563,-48.651,179.575,5.699,149.135
C01268=1125.088,-35.314,-48.662,179.576,5.704,149.136
C01269=1125.082,-35.064,-48.674,179.576,5.708,149.137
C01270=1125.077,-34.814,-48.686,179.577,5.713,149.138
C01271=1125.073,-34.565,-48.698,179.578,5.717,149.139
C01272=1125.067,-34.349,-48.708,179.578,5.721,149.139
C01273=1125.063,-34.134,-48.718,179.579,5.726,149.140
C01274=1125.059,-33.918,-48.728,179.579,5.729,149.141
C01275=1125.054,-33.703,-48.738,179.579,5.733,149.142
C01276=1125.049,-33.488,-48.748,179.580,5.736,149.142
C01277=1125.046,-33.272,-48.758,179.580,5.741,149.143
C01278=1125.041,-33.057,-48.769,179.580,5.745,149.144
C01279=1125.036,-32.842,-48.778,179.580,5.749,149.145
C01280=1125.031,-32.592,-48.790,179.581,5.753,149.146
C01281=1125.025,-32.342,-48.803,179.581,5.757,149.146
C01282=1125.021,-32.093,-48.814,179.581,5.762,149.147
C01283=1125.015,-31.843,-48.826,179.581,5.766,149.148
C01284=1125.010,-31.593,-48.838,179.581,5.770,149.149
C01285=1125.005,-31.343,-48.849,179.581,5.775,149.150
C01286=1125.000,-31.094,-48.862,179.581,5.779,149.151
C01287=1124.995,-30.844,-48.873,179.581,5.783,149.152
C01288=1124.989,-30.594,-48.885,179.581,5.787,149.153
C01289=1124.985,-30.344,-48.897,179.581,5.792,149.154
C01290=1124.979,-30.095,-48.909,179.581,5.796,149.155
C01291=1124.973,-29.846,-48.921,179.580,5.800,149.156
C01292=1124.968,-29.596,-48.933,179.580,5.804,149.157
C01293=1124.963,-29.346,-48.944,179.580,5.808,149.158
C01294=1124.958,-29.097,-48.957,179.579,5.812,149.159
C01295=1124.953,-28.847,-48.968,179.579,5.816,149.160
C01296=1124.947,-28.597,-48.980,179.578,5.820,149.161
C01297=1124.943,-28.347,-48.992,179.577,5.824,149.162
C01298=1124.937,-28.098,-49.004,179.577,5.828,149.163
C01299=1124.932,-27.848,-49.016,179.576,5.832,149.164
C01300=1124.927,-27.598,-49.028,179.575,5.836,149.165
C01301=1124.921,-27.349,-49.041,179.574,5.840,149.167
C01302=1124.917,-27.099,-49.052,179.574,5.845,149.168
C01303=1124.911,-26.849,-49.064,179.573,5.848,149.169
C01304=1124.906,-26.599,-49.076,179.572,5.852,149.170
C01305=1124.901,-26.350,-49.088,179.571,5.856,149.171
C01306=1124.895,-26.100,-49.100,179.570,5.860,149.172
C01307=1124.891,-25.851,-49.111,179.570,5.864,149.173
C01308=1124.886,-25.601,-49.124,179.571,5.870,149.174
C01309=1124.880,-25.351,-49.136,179.572,5.874,149.175
C01310=1124.875,-25.101,-49.148,179.572,5.879,149.176
C01311=1124.870,-24.852,-49.160,179.573,5.885,149.177
C01312=1124.864,-24.602,-49.172,179.574,5.889,149.178
C01313=1124.860,-24.353,-49.184,179.575,5.894,149.178
C01314=1124.854,-24.103,-49.196,179.576,5.899,149.179
C01315=1124.849,-23.853,-49.208,179.576,5.904,149.180
C01316=1124.844,-23.604,-49.221,179.577,5.909,149.181
C01317=1124.838,-23.354,-49.233,179.577,5.914,149.182
C01318=1124.833,-23.105,-49.245,179.578,5.919,149.183
C01319=1124.828,-22.855,-49.257,179.579,5.923,149.183
C01320=1124.823,-22.605,-49.270,179.580,5.928,149.184
C01321=1124.817,-22.355,-49.282,179.581,5.934,149.185
C01322=1124.812,-22.106,-49.294,179.581,5.938,149.186
C01323=1124.807,-21.856,-49.305,179.582,5.943,149.187
C01324=1124.802,-21.607,-49.318,179.583,5.948,149.188
C01325=1124.797,-21.357,-49.330,179.584,5.953,149.189
C01326=1124.792,-21.108,-49.342,179.584,5.958,149.189
C01327=1124.786,-20.858,-49.354,179.585,5.963,149.190
C01328=1124.782,-20.642,-49.365,179.586,5.967,149.191
C01329=1124.777,-20.427,-49.375,179.586,5.970,149.192
C01330=1124.773,-20.211,-49.386,179.587,5.975,149.192
C01331=1124.768,-19.997,-49.398,179.587,5.979,149.193
C01332=1124.764,-19.781,-49.408,179.588,5.983,149.194
C01333=1124.759,-19.566,-49.419,179.589,5.987,149.195
C01334=1124.755,-19.350,-49.430,179.589,5.991,149.195
C01335=1124.751,-19.135,-49.440,179.590,5.996,149.196
C01336=1124.745,-18.886,-49.452,179.591,6.000,149.197
C01337=1124.740,-18.636,-49.464,179.591,6.005,149.198
C01338=1124.735,-18.387,-49.477,179.592,6.010,149.199
C01339=1124.730,-18.137,-49.489,179.593,6.015,149.199
C01340=1124.725,-17.887,-49.502,179.594,6.019,149.200
C01341=1124.720,-17.637,-49.514,179.594,6.024,149.201
C01342=1124.714,-17.388,-49.527,179.595,6.029,149.202
C01343=1124.709,-17.138,-49.539,179.596,6.033,149.203
C01344=1124.703,-16.889,-49.552,179.596,6.038,149.203
C01345=1124.698,-16.639,-49.564,179.597,6.043,149.204
C01346=1124.693,-16.389,-49.576,179.598,6.048,149.205
C01347=1124.688,-16.139,-49.589,179.599,6.053,149.206
C01348=1124.683,-15.890,-49.602,179.599,6.057,149.207
C01349=1124.678,-15.641,-49.614,179.600,6.062,149.208
C01350=1124.673,-15.391,-49.626,179.601,6.066,149.208
C01351=1124.668,-15.141,-49.639,179.601,6.071,149.209
C01352=1124.662,-14.891,-49.652,179.602,6.076,149.210
C01353=1124.657,-14.642,-49.665,179.603,6.080,149.211
C01354=1124.652,-14.392,-49.677,179.603,6.085,149.212
C01355=1124.647,-14.142,-49.690,179.604,6.090,149.213
C01356=1124.641,-13.893,-49.702,179.605,6.094,149.213
C01357=1124.637,-13.643,-49.715,179.606,6.100,149.214
C01358=1124.632,-13.394,-49.728,179.606,6.104,149.215
C01359=1124.626,-13.144,-49.741,179.607,6.109,149.216
C01360=1124.621,-12.894,-49.753,179.608,6.113,149.217
C01361=1124.615,-12.645,-49.765,179.608,6.118,149.217
C01362=1124.611,-12.395,-49.778,179.609,6.122,149.218
C01363=1124.606,-12.146,-49.791,179.610,6.127,149.219
C01364=1124.600,-11.896,-49.804,179.610,6.132,149.220
C01365=1124.595,-11.647,-49.817,179.611,6.136,149.221
C01366=1124.590,-11.397,-49.830,179.612,6.141,149.221
C01367=1124.585,-11.147,-49.842,179.612,6.146,149.222
C01368=1124.580,-10.898,-49.855,179.613,6.150,149.223
C01369=1124.575,-10.648,-49.869,179.614,6.155,149.224
C01370=1124.570,-10.398,-49.881,179.614,6.160,149.225
C01371=1124.565,-10.149,-49.894,179.615,6.164,149.225
C01372=1124.559,-9.900,-49.906,179.616,6.169,149.226
C01373=1124.554,-9.649,-49.920,179.616,6.173,149.227
C01374=1124.549,-9.400,-49.932,179.617,6.178,149.228
C01375=1124.544,-9.151,-49.945,179.618,6.182,149.229
C01376=1124.539,-8.900,-49.959,179.618,6.187,149.230
C01377=1124.534,-8.651,-49.971,179.619,6.191,149.230
C01378=1124.528,-8.402,-49.984,179.620,6.196,149.231
C01379=1124.523,-8.151,-49.997,179.620,6.201,149.232
C01380=1124.518,-7.902,-50.010,179.621,6.205,149.233
C01381=1124.513,-7.653,-50.023,179.622,6.210,149.234
C01382=1124.508,-7.402,-50.036,179.622,6.215,149.234
C01383=1124.502,-7.153,-50.049,179.623,6.218,149.235
C01384=1124.498,-6.939,-50.060,179.623,6.223,149.236
C01385=1124.493,-6.723,-50.071,179.623,6.227,149.237
C01386=1124.489,-6.507,-50.083,179.624,6.231,149.237
C01387=1124.484,-6.292,-50.093,179.625,6.234,149.238
C01388=1124.481,-6.077,-50.104,179.625,6.238,149.239
C01389=1124.476,-5.862,-50.116,179.626,6.242,149.239
C01390=1124.471,-5.647,-50.127,179.626,6.246,149.240
C01391=1124.467,-5.432,-50.138,179.627,6.251,149.241
C01392=1124.461,-5.182,-50.152,179.628,6.254,149.242
C01393=1124.457,-4.932,-50.165,179.628,6.259,149.242
C01394=1124.452,-4.683,-50.177,179.629,6.264,149.243
C01395=1124.447,-4.433,-50.191,179.630,6.268,149.244
C01396=1124.442,-4.184,-50.204,179.630,6.273,149.245
C01397=1124.436,-3.934,-50.217,179.631,6.277,149.246
C01398=1124.431,-3.684,-50.230,179.631,6.282,149.247
C01399=1124.425,-3.434,-50.243,179.632,6.286,149.247
C01400=1124.421,-3.185,-50.257,179.633,6.291,149.248
C01401=1124.415,-2.935,-50.270,179.633,6.296,149.249
C01402=1124.410,-2.686,-50.283,179.634,6.299,149.250
C01403=1124.406,-2.436,-50.296,179.634,6.304,149.251
C01404=1124.400,-2.187,-50.310,179.635,6.309,149.251
C01405=1124.395,-1.937,-50.323,179.635,6.314,149.252
C01406=1124.390,-1.687,-50.336,179.636,6.318,149.253
C01407=1124.385,-1.438,-50.350,179.637,6.323,149.254
C01408=1124.380,-1.188,-50.363,179.637,6.327,149.255
C01409=1124.374,-0.939,-50.375,179.638,6.331,149.255
C01410=1124.369,-0.689,-50.389,179.638,6.336,149.256
C01411=1124.364,-0.440,-50.402,179.639,6.340,149.257
C01412=1124.359,-0.190,-50.416,179.639,6.345,149.258
C01413=1124.353,0.060,-50.429,179.640,6.349,149.259
C01414=1124.349,0.309,-50.443,179.641,6.354,149.260
C01415=1124.343,0.559,-50.456,179.641,6.359,149.261
C01416=1124.339,0.808,-50.470,179.641,6.363,149.261
C01417=1124.333,1.058,-50.483,179.642,6.367,149.262
C01418=1124.329,1.308,-50.496,179.643,6.372,149.263
C01419=1124.323,1.557,-50.510,179.643,6.377,149.264
C01420=1124.318,1.807,-50.523,179.644,6.381,149.265
C01421=1124.313,2.056,-50.537,179.644,6.386,149.266
C01422=1124.308,2.306,-50.550,179.645,6.390,149.266
C01423=1124.303,2.555,-50.563,179.645,6.394,149.267
C01424=1124.298,2.805,-50.577,179.646,6.399,149.268
C01425=1124.292,3.055,-50.590,179.646,6.404,149.269
C01426=1124.288,3.304,-50.604,179.647,6.408,149.270
C01427=1124.282,3.554,-50.617,179.647,6.412,149.270
C01428=1124.277,3.804,-50.631,179.648,6.417,149.271
C01429=1124.272,4.053,-50.644,179.648,6.421,149.272
C01430=1124.267,4.303,-50.658,179.649,6.426,149.273
C01431=1124.261,4.552,-50.671,179.649,6.431,149.274
C01432=1124.257,4.802,-50.685,179.649,6.435,149.275
C01433=1124.251,5.052,-50.698,179.650,6.439,149.276
C01434=1124.246,5.301,-50.712,179.651,6.444,149.276
C01435=1124.241,5.551,-50.726,179.651,6.449,149.277
C01436=1124.236,5.800,-50.739,179.652,6.453,149.278
C01437=1124.231,6.050,-50.753,179.652,6.457,149.279
C01438=1124.226,6.299,-50.766,179.652,6.462,149.280
C01439=1124.221,6.549,-50.781,179.653,6.467,149.281
C01440=1124.216,6.764,-50.792,179.653,6.470,149.281
C01441=1124.212,6.979,-50.804,179.654,6.474,149.282
C01442=1124.207,7.194,-50.815,179.654,6.478,149.283
C01443=1124.203,7.409,-50.827,179.655,6.482,149.284
C01444=1124.198,7.625,-50.839,179.655,6.486,149.285
C01445=1124.194,7.840,-50.851,179.656,6.490,149.285
C01446=1124.190,8.055,-50.863,179.656,6.494,149.286
C01447=1124.186,8.269,-50.875,179.656,6.498,149.287
C01448=1124.180,8.520,-50.888,179.657,6.502,149.287
C01449=1124.175,8.769,-50.902,179.658,6.507,149.288
C01450=1124.170,9.018,-50.916,179.659,6.512,149.289
C01451=1124.165,9.268,-50.929,179.660,6.517,149.290
C01452=1124.160,9.517,-50.943,179.660,6.521,149.291
C01453=1124.155,9.767,-50.958,179.661,6.526,149.292
C01454=1124.150,10.018,-50.971,179.662,6.530,149.292
C01455=1124.144,10.267,-50.985,179.662,6.535,149.293
C01456=1124.140,10.516,-50.999,179.663,6.540,149.294
C01457=1124.135,10.766,-51.013,179.665,6.545,149.295
C01458=1124.129,11.015,-51.026,179.665,6.550,149.295
C01459=1124.124,11.265,-51.040,179.666,6.554,149.296
C01460=1124.119,11.515,-51.055,179.667,6.559,149.297
C01461=1124.113,11.764,-51.069,179.667,6.563,149.298
C01462=1124.109,12.013,-51.082,179.668,6.568,149.299
C01463=1124.104,12.263,-51.096,179.669,6.572,149.299
C01464=1124.098,12.512,-51.110,179.670,6.577,149.300
C01465=1124.093,12.762,-51.124,179.671,6.582,149.301
C01466=1124.089,13.012,-51.138,179.672,6.587,149.302
C01467=1124.083,13.261,-51.152,179.673,6.591,149.302
C01468=1124.078,13.511,-51.167,179.674,6.596,149.303
C01469=1124.073,13.760,-51.181,179.674,6.600,149.304
C01470=1124.068,14.011,-51.194,179.675,6.605,149.305
C01471=1124.063,14.259,-51.208,179.676,6.609,149.306
C01472=1124.058,14.509,-51.222,179.677,6.614,149.306
C01473=1124.053,14.759,-51.236,179.678,6.619,149.307
C01474=1124.048,15.008,-51.251,179.679,6.623,149.308
C01475=1124.043,15.257,-51.264,179.680,6.628,149.309
C01476=1124.038,15.507,-51.279,179.681,6.632,149.309
C01477=1124.033,15.757,-51.293,179.681,6.637,149.310
C01478=1124.028,16.007,-51.307,179.682,6.642,149.311
C01479=1124.022,16.256,-51.321,179.683,6.646,149.312
C01480=1124.017,16.505,-51.335,179.684,6.651,149.312
C01481=1124.012,16.755,-51.350,179.685,6.655,149.313
C01482=1124.007,17.005,-51.364,179.685,6.660,149.314
C01483=1124.002,17.254,-51.378,179.687,6.665,149.314
C01484=1123.997,17.503,-51.392,179.688,6.669,149.315
C01485=1123.992,17.753,-51.406,179.689,6.674,149.316
C01486=1123.987,18.003,-51.421,179.690,6.678,149.317
C01487=1123.982,18.253,-51.435,179.690,6.683,149.318
C01488=1123.976,18.502,-51.449,179.691,6.687,149.318
C01489=1123.971,18.751,-51.463,179.692,6.691,149.319
C01490=1123.966,19.001,-51.477,179.693,6.696,149.320
C01491=1123.962,19.250,-51.492,179.694,6.700,149.320
C01492=1123.957,19.500,-51.507,179.695,6.705,149.321
C01493=1123.951,19.749,-51.521,179.696,6.709,149.322
C01494=1123.946,19.999,-51.536,179.697,6.714,149.323
C01495=1123.941,20.249,-51.550,179.698,6.718,149.323
C01496=1123.937,20.463,-51.562,179.699,6.722,149.324
C01497=1123.932,20.679,-51.574,179.699,6.726,149.325
C01498=1123.928,20.893,-51.587,179.700,6.730,149.325
C01499=1123.923,21.109,-51.599,179.701,6.734,149.326
C01500=1123.919,21.324,-51.612,179.702,6.738,149.326
C01501=1123.915,21.539,-51.625,179.703,6.741,149.327
C01502=1123.910,21.754,-51.636,179.704,6.746,149.328
C01503=1123.906,21.969,-51.649,179.704,6.749,149.328
C01504=1123.901,22.219,-51.664,179.705,6.753,149.329
C01505=1123.896,22.468,-51.678,179.707,6.759,149.330
C01506=1123.891,22.717,-51.693,179.707,6.763,149.330
C01507=1123.886,22.967,-51.707,179.708,6.768,149.331
C01508=1123.881,23.217,-51.722,179.709,6.772,149.332
C01509=1123.876,23.467,-51.736,179.710,6.776,149.332
C01510=1123.870,23.715,-51.751,179.711,6.781,149.333
C01511=1123.865,23.965,-51.765,179.712,6.785,149.334
C01512=1123.861,24.215,-51.779,179.713,6.790,149.335
C01513=1123.855,24.464,-51.795,179.714,6.794,149.335
C01514=1123.850,24.714,-51.809,179.715,6.798,149.336
C01515=1123.845,24.963,-51.824,179.716,6.803,149.336
C01516=1123.841,25.212,-51.839,179.717,6.807,149.337
C01517=1123.835,25.463,-51.853,179.718,6.811,149.338
C01518=1123.830,25.712,-51.868,179.719,6.816,149.339
C01519=1123.825,25.961,-51.883,179.720,6.820,149.339
C01520=1123.820,26.211,-51.897,179.721,6.824,149.340
C01521=1123.815,26.460,-51.913,179.722,6.829,149.341
C01522=1123.810,26.710,-51.927,179.723,6.833,149.341
C01523=1123.805,26.959,-51.942,179.724,6.837,149.342
C01524=1123.800,27.209,-51.957,179.725,6.842,149.343
C01525=1123.795,27.459,-51.971,179.726,6.846,149.343
C01526=1123.790,27.708,-51.986,179.727,6.850,149.344
C01527=1123.785,27.958,-52.000,179.728,6.855,149.344
C01528=1123.780,28.207,-52.016,179.729,6.859,149.345
C01529=1123.775,28.457,-52.030,179.730,6.864,149.346
C01530=1123.770,28.706,-52.045,179.731,6.868,149.347
C01531=1123.764,28.956,-52.060,179.732,6.872,149.347
C01532=1123.760,29.205,-52.075,179.733,6.877,149.348
C01533=1123.755,29.455,-52.089,179.734,6.881,149.349
C01534=1123.749,29.704,-52.105,179.735,6.885,149.349
C01535=1123.744,29.954,-52.119,179.736,6.890,149.350
C01536=1123.739,30.203,-52.135,179.737,6.894,149.351
C01537=1123.734,30.452,-52.150,179.739,6.898,149.351
C01538=1123.729,30.702,-52.164,179.740,6.903,149.352
C01539=1123.724,30.951,-52.180,179.741,6.907,149.352
C01540=1123.719,31.201,-52.194,179.742,6.911,149.353
C01541=1123.714,31.451,-52.209,179.743,6.915,149.354
C01542=1123.709,31.700,-52.224,179.744,6.920,149.354
C01543=1123.704,31.949,-52.239,179.745,6.924,149.355
C01544=1123.699,32.199,-52.254,179.746,6.928,149.356
C01545=1123.694,32.448,-52.269,179.747,6.933,149.356
C01546=1123.688,32.698,-52.284,179.748,6.937,149.357
C01547=1123.684,32.947,-52.299,179.750,6.941,149.357
C01548=1123.679,33.197,-52.315,179.751,6.945,149.358
C01549=1123.674,33.447,-52.329,179.752,6.950,149.359
C01550=1123.669,33.696,-52.345,179.753,6.954,149.359
C01551=1123.664,33.945,-52.360,179.754,6.958,149.360
C01552=1123.659,34.160,-52.373,179.755,6.963,149.361
C01553=1123.655,34.375,-52.386,179.756,6.966,149.361
C01554=1123.650,34.590,-52.399,179.757,6.970,149.362
C01555=1123.646,34.806,-52.412,179.758,6.973,149.362
C01556=1123.642,35.020,-52.425,179.759,6.977,149.363
C01557=1123.638,35.235,-52.438,179.760,6.981,149.363
C01558=1123.633,35.450,-52.451,179.760,6.984,149.364
C01559=1123.629,35.665,-52.464,179.762,6.988,149.364
C01560=1123.623,35.914,-52.480,179.763,6.992,149.365
C01561=1123.619,36.165,-52.495,179.764,6.997,149.366
C01562=1123.614,36.414,-52.510,179.765,7.001,149.366
C01563=1123.609,36.663,-52.525,179.767,7.005,149.367
C01564=1123.604,36.912,-52.541,179.768,7.009,149.367
C01565=1123.599,37.162,-52.556,179.769,7.013,149.368
C01566=1123.594,37.411,-52.571,179.770,7.018,149.369
C01567=1123.589,37.661,-52.587,179.771,7.022,149.369
C01568=1123.584,37.911,-52.602,179.772,7.026,149.370
C01569=1123.578,38.160,-52.617,179.773,7.030,149.370
C01570=1123.574,38.409,-52.632,179.774,7.035,149.371
C01571=1123.568,38.659,-52.648,179.776,7.039,149.372
C01572=1123.564,38.909,-52.664,179.777,7.043,149.372
C01573=1123.559,39.158,-52.679,179.777,7.047,149.373
C01574=1123.554,39.407,-52.694,179.779,7.051,149.373
C01575=1123.548,39.657,-52.710,179.780,7.055,149.374
C01576=1123.544,39.906,-52.725,179.781,7.059,149.375
C01577=1123.539,40.156,-52.741,179.782,7.064,149.375
C01578=1123.533,40.405,-52.756,179.783,7.068,149.376
C01579=1123.529,40.654,-52.771,179.784,7.072,149.376
C01580=1123.523,40.904,-52.787,179.786,7.076,149.377
C01581=1123.519,41.154,-52.803,179.787,7.080,149.378
C01582=1123.513,41.403,-52.818,179.788,7.084,149.378
C01583=1123.509,41.652,-52.833,179.789,7.089,149.379
C01584=1123.503,41.902,-52.849,179.790,7.093,149.379
C01585=1123.498,42.152,-52.865,179.792,7.097,149.380
C01586=1123.494,42.401,-52.880,179.793,7.101,149.381
C01587=1123.488,42.650,-52.896,179.794,7.106,149.381
C01588=1123.483,42.900,-52.911,179.795,7.110,149.382
C01589=1123.478,43.149,-52.928,179.797,7.114,149.382
C01590=1123.474,43.398,-52.943,179.798,7.118,149.383
C01591=1123.468,43.648,-52.958,179.799,7.122,149.384
C01592=1123.464,43.898,-52.974,179.800,7.126,149.384
C01593=1123.458,44.147,-52.990,179.801,7.131,149.385
C01594=1123.453,44.397,-53.006,179.802,7.135,149.385
C01595=1123.449,44.646,-53.021,179.804,7.139,149.386
C01596=1123.444,44.895,-53.037,179.805,7.143,149.386
C01597=1123.438,45.145,-53.053,179.806,7.147,149.387
C01598=1123.434,45.395,-53.069,179.807,7.151,149.387
C01599=1123.428,45.644,-53.084,179.808,7.155,149.388
C01600=1123.423,45.894,-53.100,179.809,7.159,149.389
C01601=1123.419,46.143,-53.116,179.811,7.163,149.389
C01602=1123.414,46.392,-53.132,179.812,7.167,149.390
C01603=1123.408,46.641,-53.147,179.813,7.171,149.390
C01604=1123.404,46.892,-53.163,179.815,7.176,149.391
C01605=1123.398,47.140,-53.179,179.816,7.180,149.392
C01606=1123.393,47.390,-53.195,179.817,7.184,149.392
C01607=1123.388,47.640,-53.211,179.818,7.188,149.393
C01608=1123.384,47.854,-53.225,179.819,7.191,149.393
C01609=1123.380,48.069,-53.239,179.821,7.195,149.393
C01610=1123.376,48.284,-53.252,179.821,7.199,149.394
C01611=1123.371,48.499,-53.265,179.823,7.203,149.395
C01612=1123.368,48.714,-53.280,179.824,7.206,149.395
C01613=1123.362,48.929,-53.293,179.825,7.209,149.395
C01614=1123.358,49.143,-53.307,179.826,7.213,149.396
C01615=1123.354,49.358,-53.321,179.827,7.216,149.396
C01616=1123.349,49.608,-53.337,179.828,7.220,149.397
C01617=1123.344,49.858,-53.352,179.829,7.225,149.398
C01618=1123.339,50.106,-53.369,179.831,7.228,149.398
C01619=1123.334,50.357,-53.385,179.832,7.233,149.399
C01620=1123.329,50.605,-53.401,179.833,7.237,149.399
C01621=1123.324,50.855,-53.417,179.835,7.241,149.400
C01622=1123.319,51.104,-53.433,179.836,7.245,149.400
C01623=1123.314,51.354,-53.449,179.837,7.249,149.401
C01624=1123.309,51.603,-53.466,179.838,7.253,149.401
C01625=1123.304,51.853,-53.481,179.840,7.257,149.402
C01626=1123.300,52.102,-53.498,179.841,7.262,149.403
C01627=1123.294,52.351,-53.513,179.842,7.266,149.403
C01628=1123.290,52.601,-53.530,179.843,7.269,149.404
C01629=1123.284,52.850,-53.546,179.844,7.273,149.404
C01630=1123.280,53.100,-53.562,179.846,7.277,149.405
C01631=1123.274,53.349,-53.578,179.847,7.281,149.405
C01632=1123.270,53.599,-53.595,179.848,7.286,149.406
C01633=1123.265,53.848,-53.610,179.850,7.289,149.406
C01634=1123.260,54.098,-53.627,179.851,7.294,149.407
C01635=1123.255,54.347,-53.642,179.852,7.298,149.407
C01636=1123.250,54.596,-53.659,179.853,7.302,149.408
C01637=1123.244,54.846,-53.676,179.855,7.306,149.408
C01638=1123.240,55.096,-53.692,179.856,7.310,149.409
C01639=1123.235,55.344,-53.708,179.858,7.314,149.409
C01640=1123.230,55.595,-53.724,179.859,7.318,149.410
C01641=1123.225,55.843,-53.741,179.860,7.322,149.410
C01642=1123.220,56.093,-53.757,179.861,7.327,149.411
C01643=1123.215,56.342,-53.773,179.863,7.330,149.412
C01644=1123.210,56.592,-53.789,179.864,7.334,149.412
C01645=1123.205,56.841,-53.806,179.865,7.338,149.413
C01646=1123.200,57.090,-53.823,179.867,7.342,149.413
C01647=1123.195,57.340,-53.839,179.868,7.346,149.414
C01648=1123.190,57.589,-53.855,179.869,7.350,149.414
C01649=1123.186,57.839,-53.872,179.870,7.354,149.415
C01650=1123.180,58.088,-53.888,179.872,7.358,149.415
C01651=1123.175,58.338,-53.905,179.873,7.363,149.416
C01652=1123.170,58.587,-53.921,179.875,7.366,149.416
C01653=1123.166,58.836,-53.938,179.876,7.370,149.417
C01654=1123.161,59.086,-53.954,179.877,7.375,149.417
C01655=1123.155,59.335,-53.971,179.879,7.379,149.418
C01656=1123.150,59.585,-53.987,179.880,7.383,149.418
C01657=1123.145,59.834,-54.004,179.881,7.387,149.419
C01658=1123.141,60.083,-54.020,179.883,7.391,149.419
C01659=1123.136,60.333,-54.038,179.884,7.394,149.420
C01660=1123.131,60.582,-54.054,179.885,7.398,149.420
C01661=1123.126,60.832,-54.070,179.886,7.402,149.421
C01662=1123.121,61.082,-54.087,179.888,7.406,149.421
C01663=1123.116,61.330,-54.103,179.889,7.410,149.422
C01664=1123.112,61.545,-54.117,179.891,7.414,149.422
C01665=1123.107,61.759,-54.132,179.892,7.417,149.423
C01666=1123.103,61.974,-54.146,179.893,7.420,149.423
C01667=1123.099,62.190,-54.161,179.894,7.425,149.424
C01668=1123.095,62.404,-54.175,179.895,7.428,149.424
C01669=1123.090,62.619,-54.190,179.896,7.432,149.425
C01670=1123.086,62.833,-54.204,179.897,7.435,149.425
C01671=1123.082,63.048,-54.219,179.898,7.438,149.425
C01672=1123.077,63.298,-54.235,179.900,7.442,149.426
C01673=1123.072,63.547,-54.252,179.901,7.446,149.426
C01674=1123.067,63.797,-54.269,179.902,7.450,149.427
C01675=1123.063,64.046,-54.286,179.904,7.454,149.427
C01676=1123.057,64.295,-54.302,179.906,7.458,149.428
C01677=1123.052,64.545,-54.319,179.907,7.462,149.428
C01678=1123.048,64.794,-54.336,179.908,7.466,149.429
C01679=1123.043,65.044,-54.353,179.910,7.470,149.429
C01680=1123.038,65.293,-54.369,179.911,7.474,149.430
C01681=1123.032,65.542,-54.387,179.913,7.478,149.430
C01682=1123.028,65.792,-54.403,179.914,7.482,149.431
C01683=1123.022,66.041,-54.420,179.915,7.486,149.431
C01684=1123.018,66.291,-54.437,179.917,7.490,149.432
C01685=1123.013,66.540,-54.454,179.918,7.494,149.432
C01686=1123.008,66.789,-54.471,179.919,7.498,149.433
C01687=1123.003,67.038,-54.488,179.920,7.502,149.433
C01688=1122.998,67.288,-54.505,179.922,7.505,149.434
C01689=1122.993,67.537,-54.522,179.923,7.510,149.435
C01690=1122.988,67.787,-54.539,179.925,7.514,149.435
C01691=1122.984,68.037,-54.556,179.926,7.518,149.435
C01692=1122.978,68.285,-54.573,179.927,7.522,149.436
C01693=1122.974,68.534,-54.590,179.929,7.526,149.436
C01694=1122.968,68.784,-54.607,179.931,7.530,149.437
C01695=1122.964,69.034,-54.624,179.932,7.534,149.438
C01696=1122.959,69.284,-54.641,179.933,7.538,149.438
C01697=1122.954,69.532,-54.658,179.935,7.542,149.438
C01698=1122.949,69.782,-54.675,179.936,7.546,149.439
C01699=1122.944,70.031,-54.693,179.937,7.550,149.439
C01700=1122.939,70.281,-54.709,179.939,7.554,149.440
C01701=1122.934,70.530,-54.727,179.941,7.558,149.440
C01702=1122.929,70.779,-54.744,179.942,7.562,149.441
C01703=1122.924,71.029,-54.761,179.943,7.566,149.441
C01704=1122.920,71.277,-54.778,179.944,7.569,149.442
C01705=1122.914,71.527,-54.796,179.946,7.573,149.442
C01706=1122.909,71.777,-54.813,179.947,7.577,149.443
C01707=1122.905,72.026,-54.830,179.949,7.581,149.443
C01708=1122.900,72.276,-54.847,179.950,7.585,149.444
C01709=1122.895,72.524,-54.864,179.952,7.589,149.444
C01710=1122.890,72.774,-54.882,179.953,7.593,149.445
C01711=1122.885,73.023,-54.899,179.954,7.597,149.445
C01712=1122.880,73.272,-54.916,179.956,7.601,149.446
C01713=1122.875,73.522,-54.934,179.958,7.605,149.446
C01714=1122.870,73.771,-54.952,179.959,7.609,149.447
C01715=1122.866,74.021,-54.968,179.960,7.613,149.447
C01716=1122.861,74.271,-54.986,179.962,7.617,149.448
C01717=1122.856,74.520,-55.004,179.963,7.621,149.448
C01718=1122.851,74.769,-55.020,179.964,7.625,149.449
C01719=1122.846,75.018,-55.038,179.966,7.629,149.449
C01720=1122.842,75.232,-55.053,179.967,7.632,149.450
C01721=1122.837,75.448,-55.068,179.969,7.636,149.450
C01722=1122.833,75.662,-55.083,179.970,7.639,149.450
C01723=1122.829,75.877,-55.099,179.971,7.642,149.451
C01724=1122.825,76.091,-55.113,179.972,7.646,149.451
C01725=1122.820,76.306,-55.128,179.973,7.649,149.452
C01726=1122.816,76.521,-55.143,179.975,7.653,149.452
C01727=1122.812,76.736,-55.159,179.976,7.656,149.452
C01728=1122.807,76.986,-55.176,179.977,7.660,149.453
C01729=1122.802,77.235,-55.194,179.978,7.664,149.454
C01730=1122.798,77.484,-55.211,179.979,7.667,149.454
C01731=1122.792,77.733,-55.228,179.980,7.671,149.455
C01732=1122.787,77.982,-55.246,179.981,7.674,149.455
C01733=1122.782,78.232,-55.263,179.982,7.679,149.456
C01734=1122.778,78.480,-55.281,179.983,7.682,149.456
C01735=1122.773,78.730,-55.299,179.984,7.686,149.457
C01736=1122.768,78.979,-55.316,179.984,7.690,149.457
C01737=1122.763,79.229,-55.334,179.986,7.693,149.458
C01738=1122.758,79.478,-55.352,179.987,7.697,149.459
C01739=1122.753,79.728,-55.369,179.988,7.701,149.459
C01740=1122.748,79.976,-55.387,179.989,7.704,149.460
C01741=1122.744,80.226,-55.405,179.990,7.708,149.460
C01742=1122.738,80.475,-55.422,179.991,7.712,149.461
C01743=1122.733,80.725,-55.440,179.992,7.716,149.461
C01744=1122.728,80.974,-55.458,179.993,7.719,149.462
C01745=1122.724,81.223,-55.476,179.994,7.723,149.462
C01746=1122.718,81.473,-55.493,179.996,7.727,149.463
C01747=1122.714,81.723,-55.511,179.996,7.730,149.463
C01748=1122.710,81.971,-55.529,179.998,7.735,149.464
C01749=1122.705,82.221,-55.547,179.999,7.738,149.464
C01750=1122.700,82.470,-55.564,180.000,7.742,149.465
C01751=1122.695,82.720,-55.582,-179.999,7.746,149.465
C01752=1122.690,82.969,-55.600,-179.998,7.749,149.466
C01753=1122.685,83.218,-55.618,-179.997,7.753,149.466
C01754=1122.680,83.467,-55.636,-179.995,7.757,149.467
C01755=1122.675,83.717,-55.653,-179.995,7.761,149.468
C01756=1122.670,83.966,-55.671,-179.993,7.765,149.468
C01757=1122.665,84.215,-55.689,-179.991,7.769,149.468
C01758=1122.660,84.464,-55.707,-179.991,7.772,149.469
C01759=1122.655,84.714,-55.725,-179.989,7.776,149.469
C01760=1122.650,84.963,-55.743,-179.988,7.780,149.470
C01761=1122.646,85.213,-55.761,-179.987,7.784,149.471
C01762=1122.641,85.462,-55.779,-179.986,7.787,149.471
C01763=1122.636,85.712,-55.797,-179.984,7.792,149.472
C01764=1122.631,85.961,-55.815,-179.983,7.795,149.472
C01765=1122.626,86.210,-55.833,-179.981,7.799,149.472
C01766=1122.621,86.459,-55.851,-179.981,7.803,149.473
C01767=1122.616,86.708,-55.869,-179.979,7.807,149.474
C01768=1122.611,86.958,-55.887,-179.978,7.811,149.474
C01769=1122.606,87.207,-55.905,-179.976,7.815,149.475
C01770=1122.602,87.457,-55.923,-179.975,7.818,149.475
C01771=1122.597,87.706,-55.941,-179.974,7.822,149.475
C01772=1122.592,87.955,-55.959,-179.972,7.826,149.476
C01773=1122.587,88.204,-55.977,-179.971,7.830,149.477
C01774=1122.582,88.453,-55.995,-179.970,7.834,149.477
C01775=1122.578,88.702,-56.013,-179.968,7.838,149.477
C01776=1122.573,88.917,-56.028,-179.967,7.841,149.478
C01777=1122.569,89.132,-56.045,-179.966,7.844,149.478
C01778=1122.565,89.346,-56.060,-179.964,7.848,149.479
C01779=1122.561,89.561,-56.076,-179.963,7.851,149.479
C01780=1122.556,89.776,-56.091,-179.962,7.854,149.480
C01781=1122.553,89.990,-56.107,-179.960,7.858,149.480
C01782=1122.549,90.205,-56.122,-179.959,7.861,149.480
C01783=1122.544,90.419,-56.138,-179.958,7.864,149.481
C01784=1122.539,90.669,-56.156,-179.957,7.868,149.481
C01785=1122.534,90.918,-56.174,-179.955,7.872,149.481
C01786=1122.530,91.167,-56.193,-179.954,7.876,149.482
C01787=1122.525,91.416,-56.211,-179.953,7.880,149.483
C01788=1122.520,91.666,-56.229,-179.951,7.884,149.483
C01789=1122.515,91.915,-56.247,-179.949,7.888,149.483
C01790=1122.510,92.165,-56.266,-179.948,7.892,149.484
C01791=1122.505,92.414,-56.284,-179.946,7.895,149.484
C01792=1122.501,92.663,-56.303,-179.945,7.899,149.485
C01793=1122.496,92.912,-56.321,-179.943,7.903,149.485
C01794=1122.491,93.162,-56.339,-179.941,7.907,149.486
C01795=1122.486,93.411,-56.358,-179.940,7.911,149.486
C01796=1122.481,93.660,-56.377,-179.938,7.915,149.486
C01797=1122.476,93.909,-56.395,-179.937,7.919,149.487
C01798=1122.472,94.159,-56.413,-179.935,7.923,149.487
C01799=1122.466,94.408,-56.432,-179.933,7.927,149.488
C01800=1122.462,94.657,-56.450,-179.932,7.930,149.488
C01801=1122.457,94.906,-56.468,-179.930,7.934,149.489
C01802=1122.452,95.156,-56.487,-179.929,7.938,149.489
C01803=1122.447,95.405,-56.506,-179.927,7.942,149.489
C01804=1122.442,95.654,-56.524,-179.925,7.946,149.490
C01805=1122.438,95.904,-56.542,-179.924,7.950,149.490
C01806=1122.432,96.153,-56.561,-179.922,7.954,149.491
C01807=1122.428,96.402,-56.579,-179.921,7.958,149.491
C01808=1122.424,96.651,-56.598,-179.919,7.961,149.491
C01809=1122.418,96.901,-56.617,-179.917,7.965,149.492
C01810=1122.413,97.150,-56.635,-179.915,7.969,149.492
C01811=1122.409,97.399,-56.654,-179.913,7.974,149.493
C01812=1122.403,97.649,-56.673,-179.911,7.978,149.493
C01813=1122.399,97.897,-56.691,-179.910,7.981,149.494
C01814=1122.394,98.147,-56.710,-179.908,7.985,149.494
C01815=1122.389,98.396,-56.729,-179.906,7.989,149.494
C01816=1122.384,98.645,-56.747,-179.905,7.993,149.495
C01817=1122.379,98.895,-56.767,-179.903,7.997,149.495
C01818=1122.374,99.144,-56.785,-179.900,8.001,149.495
C01819=1122.370,99.393,-56.804,-179.899,8.005,149.496
C01820=1122.365,99.643,-56.822,-179.897,8.009,149.496
C01821=1122.360,99.891,-56.841,-179.895,8.012,149.496
C01822=1122.355,100.141,-56.860,-179.893,8.016,149.497
C01823=1122.351,100.390,-56.879,-179.892,8.020,149.497
C01824=1122.346,100.639,-56.898,-179.889,8.024,149.497
C01825=1122.341,100.889,-56.916,-179.888,8.028,149.498
C01826=1122.336,101.137,-56.936,-179.886,8.032,149.498
C01827=1122.331,101.387,-56.954,-179.884,8.035,149.499
C01828=1122.326,101.636,-56.973,-179.882,8.039,149.499
C01829=1122.322,101.885,-56.992,-179.880,8.044,149.499
C01830=1122.316,102.135,-57.011,-179.878,8.048,149.500
C01831=1122.312,102.384,-57.030,-179.876,8.051,149.500
C01832=1122.308,102.599,-57.047,-179.874,8.055,149.500
C01833=1122.304,102.813,-57.063,-179.872,8.058,149.500
C01834=1122.299,103.028,-57.079,-179.871,8.061,149.501
C01835=1122.295,103.242,-57.095,-179.869,8.065,149.501
C01836=1122.291,103.456,-57.111,-179.867,8.069,149.501
C01837=1122.287,103.671,-57.128,-179.866,8.071,149.502
C01838=1122.283,103.886,-57.145,-179.864,8.075,149.502
C01839=1122.279,104.100,-57.161,-179.862,8.079,149.502
C01840=1122.273,104.349,-57.179,-179.860,8.082,149.502
C01841=1122.269,104.599,-57.199,-179.858,8.086,149.503
C01842=1122.264,104.847,-57.218,-179.856,8.090,149.503
C01843=1122.259,105.097,-57.237,-179.854,8.094,149.503
C01844=1122.255,105.346,-57.256,-179.852,8.097,149.504
C01845=1122.250,105.595,-57.276,-179.850,8.101,149.504
C01846=1122.245,105.845,-57.295,-179.847,8.105,149.504
C01847=1122.240,106.094,-57.313,-179.845,8.109,149.504
C01848=1122.236,106.343,-57.333,-179.844,8.113,149.505
C01849=1122.230,106.592,-57.352,-179.841,8.117,149.505
C01850=1122.226,106.841,-57.371,-179.839,8.121,149.505
C01851=1122.221,107.090,-57.391,-179.836,8.125,149.505
C01852=1122.216,107.340,-57.410,-179.835,8.129,149.506
C01853=1122.211,107.588,-57.429,-179.833,8.132,149.506
